(* IEC 61131-3 sources: volt/packages/volt-lsp-iec/test-corpus/pro2193/Device/Plc Logic/Application/09 Misc/Library Manager/L_MC1P_MotionControlBasic (part 6) *)

(* ---- L_MC1P_POSPROFILER.pou ---- *)
FUNCTION_BLOCK L_MC1P_POSPROFILER
VAR_INPUT
	XEXECUTE : BOOL := FALSE;
	XAUXEXECUTE : BOOL := FALSE;
	XABORT : BOOL := FALSE;
	XPOSMODE : BOOL := FALSE;
	ROVERRIDESPEED : LREAL := 1.0;
	ROVERRIDEACC : LREAL := 1.0;
	ROVERRIDEDEC : LREAL := 1.0;
	ROVERRIDEJERKACC : LREAL := 1.0;
	ROVERRIDEJERKDEC : LREAL := 1.0;
	LRACTPOS : LREAL := 0.0;
	LRACTSPEED : LREAL := 0.0;
	LRACTACC : LREAL := 0.0;
	LRTASKCYCLE : LREAL := 0.001;
	LRINVTASKCYCLE : LREAL := 1000.0;
	XCONTINUOUSUPDATE : BOOL;
	XWAIT : BOOL;
	LRCORRECTTIMEBASE : LREAL;
	WCALCPROFILEMODE : WORD;
	WSTRETCHPROFILEMODE : WORD := 0;
	XUSESTARTJERK : BOOL;
	LRSTARTJERK : LREAL;
	XUSEEXTERNPROFILECALCULATION : BOOL;
	ITFPOSPROFILECALCULATION : L_MC1P_IPosProfileCalculation;
	XINCREASEJERKDEC : BOOL;
	LRMAXJERKAPPL : LREAL;
END_VAR
VAR_OUTPUT
	XBUSY : BOOL;
	XDONE : BOOL;
	XABORTED : BOOL;
	XERROR : BOOL;
	LRSETPOS : LREAL;
	LRSETSPEED : LREAL;
	LRSETACC : LREAL;
	LRACTPROFILEJERK : LREAL;
	DWSTATE : DWORD;
	DWPROFILETYPE : DWORD;
	XNOPROFIEUPDATE : BOOL;
END_VAR
VAR_IN_OUT
	SCPROFILEPARAMETER : L_MC1P_ProfileParameter;
END_VAR
VAR
	SCPROFILEDATA : L_MC1P_ProfileData;
	XCALCPROFILEACTIVE : BOOL;
	LREVALTIME : LREAL;
	DWSTATEOFINTERPOLATOR : DWORD;
	XFLAGEXECUTE : BOOL;
	XFLAGAUXEXECUTE : BOOL;
	XFLAGABORT : BOOL;
	SCPROFILEPARAMETERINT : L_MC1P_ProfileParameter;
	SCPROFILEPARAMETEROLD : L_MC1P_ProfileParameter;
	ROVERRIDESPEEDOLD : LREAL;
	ROVERRIDEACCOLD : LREAL;
	ROVERRIDEDECOLD : LREAL;
	ROVERRIDEJERKACCOLD : LREAL;
	ROVERRIDEJERKDECOLD : LREAL;
	XSTARTCALCPROF : BOOL;
	XVELOVEREQZERO : BOOL;
	ARG1 : LREAL;
	XEXECUTEEDGE : BOOL;
	XAUXEXECUTEEDGE : BOOL;
	XABORTEDGE : BOOL;
	XCONTINUOUSUPDATEINT : BOOL;
	SCBUFFPROFILEPARAMETER : L_MC1P_ProfileParameter;
	SCBUFFPROFILEDATA : L_MC1P_ProfileData;
	XCALCULATEBUFFER : BOOL;
	XACITVATEBUFFERRANGE : BOOL;
	SCBUFFERDATAINT : L_MC1P_BufferData;
	LRTIMEACCBUFF : LREAL;
	XCALCPROFILEFIRSTCYCLEACTIVE : BOOL;
	WCALCPROFILESTEP : WORD;
	WITERATIONCYCLESLIMIT1 : WORD := 32;
	N : WORD;
	XSEARCHTIMESACTIVE : BOOL;
	XSEARCHTIMES1_DONE : BOOL;
	XCALCPROFILEDATAACTIVE : BOOL;
	XPROFILECALCULATED : BOOL;
	SIGNOFMAXVEL : LREAL;
	S_MIN : LREAL;
	DWMINPROFILETYPE : DWORD;
	VMAXMINTRIACC1 : LREAL;
	VMAXMINTRIACC2 : LREAL;
	LRRECIPRJERKACC : LREAL;
	LRRECIPRJERKDEC : LREAL;
	INITPROFILEDATA : L_MC1P_ProfileData;
	INITPHASEDATA : L_MC1P_ProfilePhaseData;
	INITINTPROFILEDATA : L_MC1P_IntProfileData;
	SCMINPOSPROFILEDATA : L_MC1P_IntProfileData;
	SCMINPROFILEDATA0 : L_MC1P_IntProfileData;
	SCMAXPROFILEDATA0 : L_MC1P_IntProfileData;
	SCMINPROFILEDATAINT : L_MC1P_IntProfileData;
	SCMINPROFILEDATA_ACC1 : L_MC1P_IntProfileDataAcc;
	SCMINPROFILEDATA_ACC2 : L_MC1P_IntProfileDataAcc;
	MINPROFILEDATA_PH57 : L_MC1P_IntProfileDataAcc;
	PROFILEPHASE : L_MC1P_ProfilePhaseData;
	JERKACCTEMP1 : LREAL;
	JERKACCTEMP2 : LREAL;
	VELPHASE4 : LREAL;
	MINVELPHASE4 : LREAL;
	PROVISIONALPROFILE : L_MC1P_IntProfileData;
	PROVISIONALPROFILEOLD : L_MC1P_IntProfileData;
	S_PROVISIONALPROFILE : LREAL;
	LRACTPROFILETIME : LREAL;
	T5_STARTVALUE : LREAL;
	T7_STARTVALUE : LREAL;
	T5_MAXVALUE : LREAL;
	T7_MAXVALUE : LREAL;
	T5_MINVALUE : LREAL;
	T7_MINVALUE : LREAL;
	MINPOSUNIT : LREAL;
	MINPOSUNITQUADRAT : LREAL;
	ESQR : LREAL;
	DT_AE : LREAL;
	DS_AE : LREAL;
	DT_A0 : LREAL;
	DS_A0 : LREAL;
	TMP : ARRAY [1..272] OF LREAL;
	INVJ : ARRAY [1..2, 1..2] OF LREAL;
	E : ARRAY [0..2] OF LREAL;
	P : ARRAY [1..2] OF LREAL;
	T5 : ARRAY [1..2] OF LREAL;
	LRMINREFJERK : LREAL;
	XPHASE0FINISHED : BOOL;
	LRSTARTACCINT : LREAL;
	LRSTARTVELINT : LREAL;
	LRSTARTPOSINT : LREAL;
	MAXPROFILEPHASEINDEX : WORD := 7;
	ALRPROFILEACC : ARRAY [0..8] OF LREAL;
	ALRPROFILEJERK : ARRAY [0..8] OF LREAL;
	ALRPROFILEPOS : ARRAY [0..8] OF LREAL;
	ALRPROFILETIME : ARRAY [0..8] OF LREAL;
	ALRPROFILEVEL : ARRAY [0..8] OF LREAL;
	REMAININGTIMEOFPROFILE : LREAL;
	REMAININGTIMEOFPROFILEAVAILABLE : BOOL;
END_VAR
END_FUNCTION_BLOCK

METHOD CALCPROFILEDATA
VAR_INPUT
	LRSTARTACC : LREAL;
	LRSTARTVEL : LREAL;
	LRSTARTPOS : LREAL;
	XVELMODE : BOOL;
END_VAR
VAR_OUTPUT
	XERROR : BOOL;
	DWSTATE : DWORD;
	DWPROFILETYPE : DWORD;
END_VAR
VAR_IN_OUT
	SCPROFILEDATA : L_MC1P_ProfileData;
	SCPROFILEPARAMETER : L_MC1P_ProfileParameter;
END_VAR
END_METHOD

METHOD CALCPROFILEDATACOMPLETE
VAR_INPUT
	LRSTARTACC : LREAL;
	LRSTARTVEL : LREAL;
	LRSTARTPOS : LREAL;
	XVELMODE : BOOL;
END_VAR
VAR_OUTPUT
	XERROR : BOOL;
	DWSTATE : DWORD;
	DWPROFILETYPE : DWORD;
END_VAR
VAR_IN_OUT
	SCPROFILEDATA : L_MC1P_ProfileData;
	SCPROFILEPARAMETER : L_MC1P_ProfileParameter;
END_VAR
END_METHOD

METHOD CALCSQRT : LREAL
VAR_INPUT
	ARG1 : LREAL;
END_VAR
END_METHOD

METHOD GETPROFILEIDXATPOS : WORD
VAR_INPUT
	LRPOS : LREAL;
END_VAR
VAR_IN_OUT
	SCPROFILEDATA : L_MC1P_ProfileData;
END_VAR
END_METHOD

METHOD GETSETVALUESNEXTCYCLE : BOOL
VAR_OUTPUT
	LRSETPOS : LREAL;
	LRSETSPEED : LREAL;
	LRSETACC : LREAL;
	DWSTATEOFINTERPOLATOR : DWORD;
END_VAR
END_METHOD

METHOD GETTIMEATPOS : LREAL
VAR_INPUT
	LRPOS : LREAL;
END_VAR
VAR_IN_OUT
	SCPROFILEDATA : L_MC1P_ProfileData;
END_VAR
END_METHOD

METHOD PROFILEINTERPOLATOR : BOOL
VAR_INPUT
	LREVALTIME : LREAL;
END_VAR
VAR_OUTPUT
	DWSTATE : DWORD;
	LRSETPOS : LREAL;
	LRSETVEL : LREAL;
	LRSETACC : LREAL;
END_VAR
VAR_IN_OUT
	SCPROFILEDATA : L_MC1P_ProfileData;
END_VAR
END_METHOD

METHOD REMAININGPROFILETIMEATPOS : BOOL
VAR_INPUT
	LRPROFILEPOS : LREAL;
END_VAR
VAR_OUTPUT
	LRREMAININGTIME : LREAL;
END_VAR
VAR_IN_OUT
	SCPROFILEDATA : L_MC1P_ProfileData;
END_VAR
END_METHOD

METHOD RESET
END_METHOD

METHOD RESETOUTPUT
END_METHOD

METHOD STRETCHPROFILE
VAR_INPUT
	LRTIMEBASE : LREAL;
END_VAR
VAR_IN_OUT
	SCPROFILEDATA : L_MC1P_ProfileData;
END_VAR
END_METHOD

METHOD FB_INIT : BOOL
VAR_INPUT
	BINITRETAINS : BOOL;
	BINCOPYCODE : BOOL;
END_VAR
END_METHOD

METHOD CALCULATEACCDIST : LREAL
VAR_INPUT
	LRACC : LREAL;
	LRJERK : LREAL;
	LRVEL : LREAL;
END_VAR
VAR_OUTPUT
	LRTIMEACC : LREAL;
END_VAR
END_METHOD

METHOD CALCULATEBUFFER : BOOL
VAR_INPUT
	LRACTPOS : LREAL;
	SCBUFFERDATA : L_MC1P_BufferData;
END_VAR
VAR_IN_OUT
	SCPROFILEPARAMETER : L_MC1P_ProfileParameter;
	SCPROFILEDATA : L_MC1P_ProfileData;
	SCBUFFPROFILEPARAMETER : L_MC1P_ProfileParameter;
	SCBUFFPROFILEDATA : L_MC1P_ProfileData;
END_VAR
END_METHOD

METHOD GETVELATPOS : LREAL
VAR_INPUT
	LRPOS : LREAL;
END_VAR
VAR_IN_OUT
	SCPROFILEDATA : L_MC1P_ProfileData;
END_VAR
END_METHOD

METHOD PROFILEINTERPOLATORBUFFER : BOOL
VAR_INPUT
	LREVALTIME : LREAL;
END_VAR
VAR_OUTPUT
	DWSTATE : DWORD;
	LRSETPOS : LREAL;
	LRSETVEL : LREAL;
	LRSETACC : LREAL;
END_VAR
VAR_IN_OUT
	SCPROFILEDATA1 : L_MC1P_ProfileData;
	SCPROFILEDATA2 : L_MC1P_ProfileData;
END_VAR
END_METHOD

METHOD SETBUFFERDATA
VAR_INPUT
	XENABLEBUFFER : BOOL;
	SCBUFFERDATA : L_MC1P_BufferData;
END_VAR
END_METHOD

METHOD CALCMINPOSUNIT : BOOL
VAR_INPUT
	SCMINPROFILEDATA : L_MC1P_IntProfileData;
	LRMAXVEL : LREAL;
	LRJERKACC1 : LREAL;
	LRMAXACC1 : LREAL;
	LRJERKACC2 : LREAL;
	LRMAXACC2 : LREAL;
	LRTARGETVEL : LREAL;
	LRTARGETACC : LREAL;
END_VAR
VAR_OUTPUT
	LRMINPOSUNIT : LREAL;
	LRMINVELUNIT : LREAL;
END_VAR
END_METHOD

METHOD CALCPROFILE : BOOL
VAR_INPUT
	DWPROFILETYPE : DWORD;
	LRSTARTACC : LREAL;
	LRSTARTVEL : LREAL;
	SCMINPROFILEDATA : L_MC1P_IntProfileData;
	SCMAXPROFILEDATA : L_MC1P_IntProfileData;
END_VAR
VAR_IN_OUT
	SCPROFILEPARAMETER : L_MC1P_ProfileParameter;
	SCPROFILEDATA : L_MC1P_ProfileData;
	WCHECKPROFILEMODE : WORD;
	DWSTATE : DWORD;
END_VAR
END_METHOD

METHOD CHECKPROFILEDATA
VAR_INPUT
	DWMODE : DWORD;
	LRTARGETPOS : LREAL;
	LRTARGETVEL : LREAL;
	LRTARGETACC : LREAL;
	LRJERKPHASE7 : LREAL;
END_VAR
VAR_OUTPUT
	XERROR : BOOL;
END_VAR
VAR_IN_OUT
	SCPROFILEDATA : L_MC1P_ProfileData;
END_VAR
END_METHOD

METHOD DEFPROFILEACCDEC
VAR_IN_OUT
	SCPROFILEPARAMETER : L_MC1P_ProfileParameter;
	LRSTARTACC : LREAL;
	LRSTARTVEL : LREAL;
	XVELMODE : BOOL;
END_VAR
END_METHOD

METHOD DEFPROFILEPHASE0 : BOOL
VAR_INPUT
	LRMINJERK : LREAL;
	XVELMODE : BOOL;
END_VAR
VAR_IN_OUT
	SCPROFILEPARAMETER : L_MC1P_ProfileParameter;
	LRSTARTACC : LREAL;
	LRSTARTVEL : LREAL;
	LRRECIPRJERKACC : LREAL;
	LRRECIPRJERKDEC : LREAL;
	SCPROFILEDATAPHASE0 : L_MC1P_ProfilePhaseData;
	SCMAXPROFILEDATA : L_MC1P_IntProfileData;
	SCMINPROFILEDATA : L_MC1P_IntProfileData;
	DWPROFILETYPE : DWORD;
	DWSTATE : DWORD;
END_VAR
END_METHOD

METHOD CALCMINPOSPROFILE : BOOL
VAR_INPUT
	MAXVEL : LREAL;
	MAXACC1 : LREAL;
	MAXACC2 : LREAL;
	JERKACC1 : LREAL;
	JERKACC2 : LREAL;
	MINJERK : LREAL;
	RECIPRJERKACC1 : LREAL;
	RECIPRJERKACC2 : LREAL;
	RECIPRMINJERK : LREAL;
	V0_ACC1 : LREAL;
	V0_ACC2 : LREAL;
	A0_ACC1 : LREAL;
	A0_ACC2 : LREAL;
	XVELMODE : BOOL;
END_VAR
VAR_IN_OUT
	DWMINPOSPROFILETYPE : DWORD;
	MINPOSPROFILEDATA : L_MC1P_IntProfileData;
	VMAXMINTRIACC1 : LREAL;
	VMAXMINTRIACC2 : LREAL;
END_VAR
END_METHOD

METHOD CALCMINPROFILE : BOOL
VAR_INPUT
	MAXVEL : LREAL;
	MAXACC1 : LREAL;
	MAXACC2 : LREAL;
	JERKACC1 : LREAL;
	JERKACC2 : LREAL;
	RECIPRJERKACC1 : LREAL;
	RECIPRJERKACC2 : LREAL;
	V0_ACC1 : LREAL;
	V0_ACC2 : LREAL;
	A0_ACC1 : LREAL;
	A0_ACC2 : LREAL;
	TARGETPOS : LREAL;
END_VAR
VAR_IN_OUT
	DWPROFILETYPE : DWORD;
	SCMINPROFILEDATA : L_MC1P_IntProfileData;
	SCMAXPROFILEDATA : L_MC1P_IntProfileData;
END_VAR
END_METHOD

METHOD CALCMINPROFILENEGACC : BOOL
VAR_INPUT
	V0 : LREAL;
	VE : LREAL;
	AMAX : LREAL;
	JERK : LREAL;
	JERKRECIPR : LREAL;
	A0 : LREAL;
	AE : LREAL;
END_VAR
VAR_OUTPUT
	DWPROFILETYPE : DWORD;
	PROFILEDATA_NEGACC : L_MC1P_IntProfileDataAcc;
END_VAR
END_METHOD

METHOD CALCMINPROFILENEGACCRND : BOOL
VAR_INPUT
	V0 : LREAL;
	VE : LREAL;
	AMAX : LREAL;
	JERK : LREAL;
	JERKRECIPR : LREAL;
	A0 : LREAL;
	AE : LREAL;
END_VAR
VAR_OUTPUT
	DWPROFILETYPE : DWORD;
	PROFILEDATA_NEGACC : L_MC1P_IntProfileDataAcc;
END_VAR
END_METHOD

METHOD CALCMINPROFILEPOSACC : BOOL
VAR_INPUT
	V0 : LREAL;
	VE : LREAL;
	AMAX : LREAL;
	A0 : LREAL;
	AE : LREAL;
	JERK : LREAL;
	JERKRECIPR : LREAL;
END_VAR
VAR_OUTPUT
	DWPROFILETYPE : DWORD;
	PROFILEDATA_POSACC : L_MC1P_IntProfileDataAcc;
END_VAR
END_METHOD

METHOD CALCMINTRI : BOOL
VAR_INPUT
	JERK : LREAL;
	RECIPRJERK : LREAL;
	A0 : LREAL;
	V0 : LREAL;
	MINCYCLETIME : LREAL;
END_VAR
VAR_OUTPUT
	VMAXMINTRIACC : LREAL;
	PROFILEDATA : L_MC1P_IntProfileDataAcc;
END_VAR
END_METHOD

METHOD CALCNEGPROFILEPHASE : BOOL
VAR_INPUT
	LRSTARTACC : LREAL;
	LRENDACC : LREAL;
	LRSTARTVEL : LREAL;
	LRJERK : LREAL;
	LRJERKRECIPR : LREAL;
	LRMINCYCLETIME : LREAL;
END_VAR
VAR_OUTPUT
	PROFILEPHASE : L_MC1P_ProfilePhaseData;
END_VAR
END_METHOD

METHOD CALCPROFILEPHASE : BOOL
VAR_INPUT
	LRSTARTACC : LREAL;
	LRENDACC : LREAL;
	LRSTARTVEL : LREAL;
	LRJERK : LREAL;
	LRJERKRECIPR : LREAL;
	LRMINCYCLETIME : LREAL;
END_VAR
VAR_OUTPUT
	PROFILEPHASE : L_MC1P_ProfilePhaseData;
END_VAR
END_METHOD

METHOD CALCPROVISIONALPROFILE
VAR_IN_OUT
	SCPROFILEPARAMETERINT : L_MC1P_ProfileParameter;
	LRSTARTVELINT : LREAL;
	LRSTARTACCINT : LREAL;
	LRRECIPRJERKACC : LREAL;
	LRRECIPRJERKDEC : LREAL;
	LRACTPROFILETIME : LREAL;
	XVELMODE : BOOL;
	SCPROVISIONALPROFILE : L_MC1P_IntProfileData;
END_VAR
END_METHOD

METHOD CALCPROVISIONALPROFILEDATA : BOOL
VAR_IN_OUT
	LRSTARTPOS : LREAL;
	LRSTARTVEL : LREAL;
	LRSTARTACC : LREAL;
	LRSTARTVELINT : LREAL;
	LRSTARTACCINT : LREAL;
	LRRECIPRJERKACC : LREAL;
	LRRECIPRJERKDEC : LREAL;
	SCPROFILEPARAMETERINT : L_MC1P_ProfileParameter;
	XVELMODE : BOOL;
	SIGNOFMAXVEL : LREAL;
	DWPROFILETYPE : DWORD;
	DWMINPOSPROFILETYPE : DWORD;
	XCALCPROFILE : BOOL;
	WCALCPROFILESTEP : WORD;
	XPOSITIVEMOVEMENT : BOOL;
	SCPROFILEDATAPHASE0 : L_MC1P_ProfilePhaseData;
	SCPROFILEDATA : L_MC1P_ProfileData;
	DWSTATECALCPROFILE : DWORD;
	SCMAXPROFILEDATA : L_MC1P_IntProfileData;
	SCMINPROFILEDATA : L_MC1P_IntProfileData;
END_VAR
END_METHOD

METHOD CALCREVPROFILE : BOOL
VAR_INPUT
	V0 : LREAL;
	VE : LREAL;
	AMAX : LREAL;
	A0 : LREAL;
	AE : LREAL;
	JERK : LREAL;
	JERKRECIPR : LREAL;
END_VAR
VAR_OUTPUT
	DWPROFILETYPE : DWORD;
	PROFILEDATA_POSACC : L_MC1P_IntProfileDataAcc;
END_VAR
END_METHOD

METHOD CALCVELPROFILEPHASE : BOOL
VAR_INPUT
	LRSTARTACC : LREAL;
	LRENDACC : LREAL;
	LRSTARTVEL : LREAL;
	LRJERK : LREAL;
	LRJERKRECIPR : LREAL;
	LRMINCYCLETIME : LREAL;
END_VAR
VAR_OUTPUT
	PROFILEPHASE : L_MC1P_ProfilePhaseData;
END_VAR
END_METHOD

METHOD IDENTINCRJERKPROFILE : BOOL
VAR_INPUT
	MINPROFILETYPE : DWORD;
	MAXACC2 : LREAL;
	MAXJERK : LREAL;
	V0_ACC1 : LREAL;
	V0_ACC2 : LREAL;
	A0_ACC1 : LREAL;
	A0_ACC2 : LREAL;
	TARGETPOS : LREAL;
END_VAR
VAR_OUTPUT
	DWINCRJERKPROFILETYPE : DWORD;
END_VAR
VAR_IN_OUT
	JERKACC2 : LREAL;
	RECIPRJERKACC2 : LREAL;
	SCMAXPROFILEDATA : L_MC1P_IntProfileData;
	SCMINPROFILEDATA : L_MC1P_IntProfileData;
END_VAR
END_METHOD

METHOD IDENTMINNEGPROFILE : BOOL
VAR_INPUT
	MINPROFILETYPE : DWORD;
	MAXVEL : LREAL;
	MAXACC : LREAL;
	JERK : LREAL;
	RECIPRJERK : LREAL;
	V0_ACC1 : LREAL;
	V0_ACC2 : LREAL;
	A0_ACC1 : LREAL;
	A0_ACC2 : LREAL;
	TARGETPOS : LREAL;
END_VAR
VAR_OUTPUT
	DWPROFILETYPE : DWORD;
END_VAR
VAR_IN_OUT
	SCMAXPROFILEDATA : L_MC1P_IntProfileData;
	SCMINPROFILEDATA : L_MC1P_IntProfileData;
END_VAR
END_METHOD

METHOD IDENTMINNEGPROFILE_A0EQ0_AENE0
VAR_INPUT
	MAXVEL : LREAL;
	SIGNOFMAXVEL : LREAL;
	MAXACC : LREAL;
	JERK : LREAL;
	RECIPRJERK : LREAL;
	V0_ACC1 : LREAL;
	V0_ACC2 : LREAL;
	A0_ACC1 : LREAL;
	A0_ACC2 : LREAL;
	TARGETPOS : LREAL;
	TARGETPOSTOLERANCE : LREAL;
END_VAR
VAR_OUTPUT
	DWPROFILETYPE : DWORD;
END_VAR
VAR_IN_OUT
	SCMAXPROFILEDATA : L_MC1P_IntProfileData;
	SCMINPROFILEDATA : L_MC1P_IntProfileData;
END_VAR
END_METHOD

METHOD IDENTMINNEGPROFILE_AENE0
VAR_INPUT
	MAXVEL : LREAL;
	SIGNOFMAXVEL : LREAL;
	MAXACC : LREAL;
	JERK : LREAL;
	RECIPRJERK : LREAL;
	V0_ACC1 : LREAL;
	V0_ACC2 : LREAL;
	A0_ACC1 : LREAL;
	A0_ACC2 : LREAL;
	TARGETPOS : LREAL;
	TARGETPOSTOLERANCE : LREAL;
END_VAR
VAR_IN_OUT
	SCMAXPROFILEDATA : L_MC1P_IntProfileData;
	SCMINPROFILEDATA : L_MC1P_IntProfileData;
	DWPROFILETYPE : DWORD;
END_VAR
END_METHOD

METHOD IDENTMINPOSPROFILE_AENE0
VAR_INPUT
	MAXVEL : LREAL;
	SIGNOFMAXVEL : LREAL;
	MAXACC : LREAL;
	JERK : LREAL;
	RECIPRJERK : LREAL;
	V0_ACC1 : LREAL;
	V0_ACC2 : LREAL;
	A0_ACC1 : LREAL;
	A0_ACC2 : LREAL;
	TARGETPOS : LREAL;
	TARGETPOSTOLERANCE : LREAL;
END_VAR
VAR_IN_OUT
	SCMAXPROFILEDATA : L_MC1P_IntProfileData;
	SCMINPROFILEDATA : L_MC1P_IntProfileData;
	DWPROFILETYPE : DWORD;
END_VAR
END_METHOD

METHOD IDENTMINPROFILE : BOOL
VAR_INPUT
	MAXVEL : LREAL;
	MAXACC1 : LREAL;
	MAXACC2 : LREAL;
	MINJERK : LREAL;
	RECIPRMINJERK : LREAL;
	V0_ACC1 : LREAL;
	A0_ACC1 : LREAL;
	TARGETPOS : LREAL;
	XVELMODE : BOOL;
END_VAR
VAR_IN_OUT
	DWPROFILETYPE : DWORD;
	SCMAXPROFILEDATA : L_MC1P_IntProfileData;
	SCMINPROFILEDATA : L_MC1P_IntProfileData;
	DWMINPROFILETYPE : DWORD;
	V0_ACC2 : LREAL;
	A0_ACC2 : LREAL;
	JERKACC1 : LREAL;
	JERKACC2 : LREAL;
	RECIPRJERKACC1 : LREAL;
	RECIPRJERKACC2 : LREAL;
	DWSTATE : DWORD;
END_VAR
END_METHOD

METHOD IDENTPROFILETYPE : DWORD
VAR_INPUT
	XVELMODE : BOOL;
	LRSTARTVEL : LREAL;
	LRSTARTACC : LREAL;
END_VAR
VAR_IN_OUT
	SCPROFILEPARAMETER : L_MC1P_ProfileParameter;
	DWPROFILETYPE : DWORD;
	SCMINPROFILEDATA : L_MC1P_IntProfileData;
	SCMAXPROFILEDATA : L_MC1P_IntProfileData;
	DWSTATE : DWORD;
END_VAR
END_METHOD

METHOD IDENTSIMPLEPROFILE
VAR_INPUT
	DWMINPOSPROFILETYPE : DWORD;
	VMAXMINTRIACC1 : LREAL;
	VMAXMINTRIACC2 : LREAL;
	MAXACC1 : LREAL;
	MAXACC2 : LREAL;
	JERKACC1 : LREAL;
	JERKACC2 : LREAL;
	V0_ACC1 : LREAL;
	A0_ACC1 : LREAL;
	RECIPRJERKACC1 : LREAL;
	RECIPRJERKACC2 : LREAL;
	LRTARGETPOS : LREAL;
	SIGNOFMAXVEL : LREAL;
END_VAR
VAR_OUTPUT
	DWPROFILETYPE : DWORD;
END_VAR
VAR_IN_OUT
	SCMINPROFILEDATA : L_MC1P_IntProfileData;
	SCMAXPROFILEDATA : L_MC1P_IntProfileData;
	V0_ACC2 : LREAL;
	A0_ACC2 : LREAL;
END_VAR
END_METHOD

METHOD IDENTSIMPLETRAPNEG : BOOL
VAR_INPUT
	MAXACC2 : LREAL;
	V0_ACC1 : LREAL;
	V0_ACC2 : LREAL;
	A0_ACC1 : LREAL;
	A0_ACC2 : LREAL;
	JERKACC1 : LREAL;
	JERKACC2 : LREAL;
	RECIPRJERKACC2 : LREAL;
	TARGETPOS : LREAL;
	SIGNOFMAXVEL : LREAL;
END_VAR
VAR_OUTPUT
	DWPROFILETYPE : DWORD;
END_VAR
VAR_IN_OUT
	SCMINPROFILEDATA : L_MC1P_IntProfileData;
	SCMAXPROFILEDATA : L_MC1P_IntProfileData;
END_VAR
END_METHOD

METHOD IDENTSIMPLETRAPPOS : BOOL
VAR_INPUT
	MAXACC1 : LREAL;
	V0_ACC1 : LREAL;
	V0_ACC2 : LREAL;
	A0_ACC1 : LREAL;
	A0_ACC2 : LREAL;
	JERKACC1 : LREAL;
	JERKACC2 : LREAL;
	RECIPRJERKACC1 : LREAL;
	TARGETPOS : LREAL;
	SIGNOFMAXVEL : LREAL;
END_VAR
VAR_OUTPUT
	DWPROFILETYPE : DWORD;
END_VAR
VAR_IN_OUT
	SCMINPROFILEDATA : L_MC1P_IntProfileData;
	SCMAXPROFILEDATA : L_MC1P_IntProfileData;
END_VAR
END_METHOD

METHOD IDENTSIMPLETRAPPOSTRINEG : BOOL
VAR_INPUT
	MAXACC1 : LREAL;
	JERKACC1 : LREAL;
	RECIPRJERKACC1 : LREAL;
	V0_ACC1 : LREAL;
	A0_ACC1 : LREAL;
	VMAXACC1 : LREAL;
	VMAXACC2 : LREAL;
	JERKACC2 : LREAL;
	TARGETPOS : LREAL;
	SIGNOFMAXVEL : LREAL;
END_VAR
VAR_OUTPUT
	DWPROFILETYPE : DWORD;
END_VAR
VAR_IN_OUT
	SCMINPROFILEDATA : L_MC1P_IntProfileData;
	SCMAXPROFILEDATA : L_MC1P_IntProfileData;
END_VAR
END_METHOD

METHOD IDENTSIMPLETRINEG : BOOL
VAR_INPUT
	V0_ACC1 : LREAL;
	A0_ACC1 : LREAL;
	A0_ACC2 : LREAL;
	JERKACC1 : LREAL;
	JERKACC2 : LREAL;
	RECIPRJERKACC2 : LREAL;
	TARGETPOS : LREAL;
	SIGNOFMAXVEL : LREAL;
END_VAR
VAR_OUTPUT
	DWPROFILETYPE : DWORD;
END_VAR
VAR_IN_OUT
	SCMINPROFILEDATA : L_MC1P_IntProfileData;
	SCMAXPROFILEDATA : L_MC1P_IntProfileData;
END_VAR
END_METHOD

METHOD IDENTSIMPLETRIPOS : BOOL
VAR_INPUT
	V0_ACC1 : LREAL;
	A0_ACC1 : LREAL;
	A0_ACC2 : LREAL;
	JERKACC1 : LREAL;
	JERKACC2 : LREAL;
	RECIPRJERKACC1 : LREAL;
	TARGETPOS : LREAL;
	SIGNOFMAXVEL : LREAL;
END_VAR
VAR_OUTPUT
	DWPROFILETYPE : DWORD;
END_VAR
VAR_IN_OUT
	SCMINPROFILEDATA : L_MC1P_IntProfileData;
	SCMAXPROFILEDATA : L_MC1P_IntProfileData;
END_VAR
END_METHOD

METHOD IDENTSIMPLETRIPOSTRAPNEG : BOOL
VAR_INPUT
	V0_ACC1 : LREAL;
	A0_ACC1 : LREAL;
	MAXACC2 : LREAL;
	JERKACC2 : LREAL;
	RECIPRJERKACC2 : LREAL;
	V0_ACC2 : LREAL;
	A0_ACC2 : LREAL;
	VMAXMINTRIACC1 : LREAL;
	JERKACC1 : LREAL;
	RECIPRJERKACC1 : LREAL;
	TARGETPOS : LREAL;
	SIGNOFMAXVEL : LREAL;
END_VAR
VAR_OUTPUT
	DWPROFILETYPE : DWORD;
END_VAR
VAR_IN_OUT
	SCMINPROFILEDATA : L_MC1P_IntProfileData;
	SCMAXPROFILEDATA : L_MC1P_IntProfileData;
END_VAR
END_METHOD

METHOD IDENTSIMPLETRIPOSTRINEG : BOOL
VAR_INPUT
	V0_ACC1 : LREAL;
	A0_ACC1 : LREAL;
	AMAX : LREAL;
	RECIPRJERKACC1 : LREAL;
	JERKACC1 : LREAL;
	JERKACC2 : LREAL;
	TARGETPOS : LREAL;
	VMAXACC1 : LREAL;
	VMAXACC2 : LREAL;
	SIGNOFMAXVEL : LREAL;
END_VAR
VAR_OUTPUT
	DWPROFILETYPE : DWORD;
END_VAR
VAR_IN_OUT
	SCMINPROFILEDATA : L_MC1P_IntProfileData;
	SCMAXPROFILEDATA : L_MC1P_IntProfileData;
END_VAR
END_METHOD

METHOD CALCPROFILE_10X0_30X0 : BOOL
VAR_INPUT
	LRSTARTACC : LREAL;
	LRSTARTVEL : LREAL;
	LRMAXACC : LREAL;
	LRMAXDEC : LREAL;
	LRMAXVEL : LREAL;
	LRTARGETACC : LREAL;
	LRTARGETVEL : LREAL;
	LRTARGETPOS : LREAL;
	LRJERKACC : LREAL;
	LRJERKDEC : LREAL;
	LRJERKTIMEACC : LREAL;
	LRJERKTIMEDEC : LREAL;
	SCMINPROFILEDATA : L_MC1P_IntProfileData;
	SCMAXPROFILEDATA : L_MC1P_IntProfileData;
END_VAR
VAR_OUTPUT
	DWSTATE : DWORD;
END_VAR
VAR_IN_OUT
	SCPROFILEDATA : L_MC1P_ProfileData;
	SCPROFILEPARAMETER : L_MC1P_ProfileParameter;
END_VAR
END_METHOD

METHOD CALCPROFILE_20CB : BOOL
VAR_INPUT
	LRSTARTACC : LREAL;
	LRSTARTVEL : LREAL;
	LRMAXACC : LREAL;
	LRMAXDEC : LREAL;
	LRMAXVEL : LREAL;
	LRTARGETACC : LREAL;
	LRTARGETVEL : LREAL;
	LRTARGETPOS : LREAL;
	LRJERKACC : LREAL;
	LRJERKDEC : LREAL;
	LRJERKTIMEACC : LREAL;
	LRJERKTIMEDEC : LREAL;
	SCMAXPROFILEDATA : L_MC1P_IntProfileData;
	SCMINPROFILEDATA : L_MC1P_IntProfileData;
END_VAR
VAR_OUTPUT
	DWSTATE : DWORD;
END_VAR
VAR_IN_OUT
	SCPROFILEDATA : L_MC1P_ProfileData;
	SCPROFILEPARAMETER : L_MC1P_ProfileParameter;
END_VAR
END_METHOD

METHOD CALCPROFILE_20CB_LINVELPH57_NEG : BOOL
VAR_INPUT
	LRSTARTACC : LREAL;
	LRSTARTVEL : LREAL;
	LRMAXACC : LREAL;
	LRMAXDEC : LREAL;
	LRMAXVEL : LREAL;
	LRTARGETACC : LREAL;
	LRTARGETVEL : LREAL;
	LRTARGETPOS : LREAL;
	LRJERKACC : LREAL;
	LRJERKDEC : LREAL;
	LRJERKTIMEACC : LREAL;
	LRJERKTIMEDEC : LREAL;
	T7 : LREAL;
END_VAR
VAR_IN_OUT
	SCPROFILEDATA : L_MC1P_ProfileData;
END_VAR
END_METHOD

METHOD CALCPROFILE_20CB_LINVELPH57_POS : BOOL
VAR_INPUT
	LRSTARTACC : LREAL;
	LRSTARTVEL : LREAL;
	LRMAXACC : LREAL;
	LRMAXDEC : LREAL;
	LRMAXVEL : LREAL;
	LRTARGETACC : LREAL;
	LRTARGETVEL : LREAL;
	LRTARGETPOS : LREAL;
	LRJERKACC : LREAL;
	LRJERKDEC : LREAL;
	LRJERKTIMEACC : LREAL;
	LRJERKTIMEDEC : LREAL;
	T7 : LREAL;
END_VAR
VAR_IN_OUT
	SCPROFILEDATA : L_MC1P_ProfileData;
END_VAR
END_METHOD

METHOD CALCPROFILE_20CB_AOGEAMAX_PROFILEDATA : BOOL
VAR_INPUT
	LRSTARTACC : LREAL;
	LRSTARTVEL : LREAL;
	LRMAXACC : LREAL;
	LRMAXDEC : LREAL;
	LRMAXVEL : LREAL;
	LRTARGETACC : LREAL;
	LRTARGETVEL : LREAL;
	LRTARGETPOS : LREAL;
	LRJERKACC : LREAL;
	LRJERKDEC : LREAL;
	LRJERKTIMEACC : LREAL;
	LRJERKTIMEDEC : LREAL;
	T7 : LREAL;
END_VAR
VAR_IN_OUT
	SCPROFILEDATA : L_MC1P_ProfileData;
END_VAR
END_METHOD

METHOD CALCPROFILE_20CB_AOGEAMAX_SEARCHTIMES : BOOL
VAR_INPUT
	LRSTARTACC : LREAL;
	LRSTARTVEL : LREAL;
	LRMAXACC : LREAL;
	LRMAXDEC : LREAL;
	LRMAXVEL : LREAL;
	LRTARGETACC : LREAL;
	LRTARGETVEL : LREAL;
	LRTARGETPOS : LREAL;
	LRJERKACC : LREAL;
	LRJERKDEC : LREAL;
	LRJERKTIMEACC : LREAL;
	LRJERKTIMEDEC : LREAL;
	T7_MINVALUE : LREAL;
	T7_MAXVALUE : LREAL;
END_VAR
VAR_IN_OUT
	T7 : LREAL;
END_VAR
END_METHOD

METHOD CALCPROFILE_20D1 : BOOL
VAR_INPUT
	LRSTARTACC : LREAL;
	LRSTARTVEL : LREAL;
	LRMAXACC : LREAL;
	LRMAXDEC : LREAL;
	LRMAXVEL : LREAL;
	LRTARGETACC : LREAL;
	LRTARGETVEL : LREAL;
	LRTARGETPOS : LREAL;
	LRJERKACC : LREAL;
	LRJERKDEC : LREAL;
	LRJERKTIMEACC : LREAL;
	LRJERKTIMEDEC : LREAL;
	SCMAXPROFILEDATA : L_MC1P_IntProfileData;
	SCMINPROFILEDATA : L_MC1P_IntProfileData;
END_VAR
VAR_OUTPUT
	DWSTATE : DWORD;
END_VAR
VAR_IN_OUT
	SCPROFILEDATA : L_MC1P_ProfileData;
END_VAR
END_METHOD

METHOD CALCPROFILE_20D1_PROFILEDATA : BOOL
VAR_INPUT
	LRSTARTACC : LREAL;
	LRSTARTVEL : LREAL;
	LRMAXACC : LREAL;
	LRMAXDEC : LREAL;
	LRMAXVEL : LREAL;
	LRTARGETACC : LREAL;
	LRTARGETVEL : LREAL;
	LRTARGETPOS : LREAL;
	LRJERKACC : LREAL;
	LRJERKDEC : LREAL;
	LRJERKTIMEACC : LREAL;
	LRJERKTIMEDEC : LREAL;
	T7 : LREAL;
END_VAR
VAR_IN_OUT
	SCPROFILEDATA : L_MC1P_ProfileData;
END_VAR
END_METHOD

METHOD CALCPROFILE_20D1_SEARCHTIMES : BOOL
VAR_INPUT
	LRSTARTACC : LREAL;
	LRSTARTVEL : LREAL;
	LRMAXACC : LREAL;
	LRMAXDEC : LREAL;
	LRMAXVEL : LREAL;
	LRTARGETACC : LREAL;
	LRTARGETVEL : LREAL;
	LRTARGETPOS : LREAL;
	LRJERKACC : LREAL;
	LRJERKDEC : LREAL;
	LRJERKTIMEACC : LREAL;
	LRJERKTIMEDEC : LREAL;
	T7_MINVALUE : LREAL;
	T7_MAXVALUE : LREAL;
END_VAR
VAR_IN_OUT
	T7 : LREAL;
END_VAR
END_METHOD

METHOD CALCPROFILE_20DB : BOOL
VAR_INPUT
	LRSTARTACC : LREAL;
	LRSTARTVEL : LREAL;
	LRMAXACC : LREAL;
	LRMAXDEC : LREAL;
	LRMAXVEL : LREAL;
	LRTARGETACC : LREAL;
	LRTARGETVEL : LREAL;
	LRTARGETPOS : LREAL;
	LRJERKACC : LREAL;
	LRJERKDEC : LREAL;
	LRJERKTIMEACC : LREAL;
	LRJERKTIMEDEC : LREAL;
	SCMAXPROFILEDATA : L_MC1P_IntProfileData;
	SCMINPROFILEDATA : L_MC1P_IntProfileData;
END_VAR
VAR_OUTPUT
	DWSTATE : DWORD;
END_VAR
VAR_IN_OUT
	SCPROFILEDATA : L_MC1P_ProfileData;
	SCPROFILEPARAMETER : L_MC1P_ProfileParameter;
END_VAR
END_METHOD

METHOD CALCPROFILE_20DB_PROFILEDATA : BOOL
VAR_INPUT
	LRSTARTACC : LREAL;
	LRSTARTVEL : LREAL;
	LRMAXACC : LREAL;
	LRMAXDEC : LREAL;
	LRMAXVEL : LREAL;
	LRTARGETACC : LREAL;
	LRTARGETVEL : LREAL;
	LRTARGETPOS : LREAL;
	LRJERKACC : LREAL;
	LRJERKDEC : LREAL;
	LRJERKTIMEACC : LREAL;
	LRJERKTIMEDEC : LREAL;
	T7 : LREAL;
END_VAR
VAR_IN_OUT
	SCPROFILEDATA : L_MC1P_ProfileData;
END_VAR
END_METHOD

METHOD CALCPROFILE_20DB_SEARCHTIMES : BOOL
VAR_INPUT
	LRSTARTACC : LREAL;
	LRSTARTVEL : LREAL;
	LRMAXACC : LREAL;
	LRMAXDEC : LREAL;
	LRMAXVEL : LREAL;
	LRTARGETACC : LREAL;
	LRTARGETVEL : LREAL;
	LRTARGETPOS : LREAL;
	LRJERKACC : LREAL;
	LRJERKDEC : LREAL;
	LRJERKTIMEACC : LREAL;
	LRJERKTIMEDEC : LREAL;
	T7_MINVALUE : LREAL;
	T7_MAXVALUE : LREAL;
END_VAR
VAR_IN_OUT
	T7 : LREAL;
END_VAR
END_METHOD

METHOD CALCPROFILE_40A0 : BOOL
VAR_INPUT
	LRSTARTACC : LREAL;
	LRSTARTVEL : LREAL;
	LRMAXACC : LREAL;
	LRMAXDEC : LREAL;
	LRMAXVEL : LREAL;
	LRTARGETACC : LREAL;
	LRTARGETVEL : LREAL;
	LRTARGETPOS : LREAL;
	LRJERKACC : LREAL;
	LRJERKDEC : LREAL;
	LRJERKTIMEACC : LREAL;
	LRJERKTIMEDEC : LREAL;
END_VAR
VAR_OUTPUT
	DWSTATE : DWORD;
END_VAR
VAR_IN_OUT
	SCPROFILEDATA : L_MC1P_ProfileData;
	SCPROFILEPARAMETER : L_MC1P_ProfileParameter;
END_VAR
END_METHOD

METHOD CALCPROFILE_40A0_LINVELPH1357_NEG : BOOL
VAR_INPUT
	LRSTARTACC : LREAL;
	LRSTARTVEL : LREAL;
	LRMAXACC : LREAL;
	LRMAXDEC : LREAL;
	LRMAXVEL : LREAL;
	LRTARGETACC : LREAL;
	LRTARGETVEL : LREAL;
	LRTARGETPOS : LREAL;
	LRJERKACC : LREAL;
	LRJERKDEC : LREAL;
	LRJERKTIMEACC : LREAL;
	LRJERKTIMEDEC : LREAL;
END_VAR
VAR_IN_OUT
	SCPROFILEDATA : L_MC1P_ProfileData;
END_VAR
END_METHOD

METHOD CALCPROFILE_40A0_LINVELPH1357_POS : BOOL
VAR_INPUT
	LRSTARTACC : LREAL;
	LRSTARTVEL : LREAL;
	LRMAXACC : LREAL;
	LRMAXDEC : LREAL;
	LRMAXVEL : LREAL;
	LRTARGETACC : LREAL;
	LRTARGETVEL : LREAL;
	LRTARGETPOS : LREAL;
	LRJERKACC : LREAL;
	LRJERKDEC : LREAL;
	LRJERKTIMEACC : LREAL;
	LRJERKTIMEDEC : LREAL;
END_VAR
VAR_IN_OUT
	SCPROFILEDATA : L_MC1P_ProfileData;
END_VAR
END_METHOD

METHOD CALCPROFILE_40A0_LINVELPH13_NEG : BOOL
VAR_INPUT
	LRSTARTACC : LREAL;
	LRSTARTVEL : LREAL;
	LRMAXACC : LREAL;
	LRMAXDEC : LREAL;
	LRMAXVEL : LREAL;
	LRTARGETACC : LREAL;
	LRTARGETVEL : LREAL;
	LRTARGETPOS : LREAL;
	LRJERKACC : LREAL;
	LRJERKDEC : LREAL;
	LRJERKTIMEACC : LREAL;
	LRJERKTIMEDEC : LREAL;
END_VAR
VAR_IN_OUT
	SCPROFILEDATA : L_MC1P_ProfileData;
END_VAR
END_METHOD

METHOD CALCPROFILE_40A0_LINVELPH13_POS : BOOL
VAR_INPUT
	LRSTARTACC : LREAL;
	LRSTARTVEL : LREAL;
	LRMAXACC : LREAL;
	LRMAXDEC : LREAL;
	LRMAXVEL : LREAL;
	LRTARGETACC : LREAL;
	LRTARGETVEL : LREAL;
	LRTARGETPOS : LREAL;
	LRJERKACC : LREAL;
	LRJERKDEC : LREAL;
	LRJERKTIMEACC : LREAL;
	LRJERKTIMEDEC : LREAL;
END_VAR
VAR_IN_OUT
	SCPROFILEDATA : L_MC1P_ProfileData;
END_VAR
END_METHOD

METHOD CALCPROFILE_40A0_LINVELPH57_NEG : BOOL
VAR_INPUT
	LRSTARTACC : LREAL;
	LRSTARTVEL : LREAL;
	LRMAXACC : LREAL;
	LRMAXDEC : LREAL;
	LRMAXVEL : LREAL;
	LRTARGETACC : LREAL;
	LRTARGETVEL : LREAL;
	LRTARGETPOS : LREAL;
	LRJERKACC : LREAL;
	LRJERKDEC : LREAL;
	LRJERKTIMEACC : LREAL;
	LRJERKTIMEDEC : LREAL;
END_VAR
VAR_IN_OUT
	SCPROFILEDATA : L_MC1P_ProfileData;
END_VAR
END_METHOD

METHOD CALCPROFILE_40A0_LINVELPH57_POS : BOOL
VAR_INPUT
	LRSTARTACC : LREAL;
	LRSTARTVEL : LREAL;
	LRMAXACC : LREAL;
	LRMAXDEC : LREAL;
	LRMAXVEL : LREAL;
	LRTARGETACC : LREAL;
	LRTARGETVEL : LREAL;
	LRTARGETPOS : LREAL;
	LRJERKACC : LREAL;
	LRJERKDEC : LREAL;
	LRJERKTIMEACC : LREAL;
	LRJERKTIMEDEC : LREAL;
END_VAR
VAR_IN_OUT
	SCPROFILEDATA : L_MC1P_ProfileData;
END_VAR
END_METHOD

METHOD CALCPROFILE_40A0_A0LTAMAX_NEG : BOOL
VAR_INPUT
	LRSTARTACC : LREAL;
	LRSTARTVEL : LREAL;
	LRMAXACC : LREAL;
	LRMAXDEC : LREAL;
	LRMAXVEL : LREAL;
	LRTARGETACC : LREAL;
	LRTARGETVEL : LREAL;
	LRTARGETPOS : LREAL;
	LRJERKACC : LREAL;
	LRJERKDEC : LREAL;
	LRJERKTIMEACC : LREAL;
	LRJERKTIMEDEC : LREAL;
END_VAR
VAR_IN_OUT
	SCPROFILEDATA : L_MC1P_ProfileData;
END_VAR
END_METHOD

METHOD CALCPROFILE_40A0_A0LTAMAX_POS : BOOL
VAR_INPUT
	LRSTARTACC : LREAL;
	LRSTARTVEL : LREAL;
	LRMAXACC : LREAL;
	LRMAXDEC : LREAL;
	LRMAXVEL : LREAL;
	LRTARGETACC : LREAL;
	LRTARGETVEL : LREAL;
	LRTARGETPOS : LREAL;
	LRJERKACC : LREAL;
	LRJERKDEC : LREAL;
	LRJERKTIMEACC : LREAL;
	LRJERKTIMEDEC : LREAL;
END_VAR
VAR_IN_OUT
	SCPROFILEDATA : L_MC1P_ProfileData;
END_VAR
END_METHOD

METHOD CALCPROFILE_40B0 : BOOL
VAR_INPUT
	LRSTARTACC : LREAL;
	LRSTARTVEL : LREAL;
	LRMAXACC : LREAL;
	LRMAXDEC : LREAL;
	LRMAXVEL : LREAL;
	LRTARGETACC : LREAL;
	LRTARGETVEL : LREAL;
	LRTARGETPOS : LREAL;
	LRJERKACC : LREAL;
	LRJERKDEC : LREAL;
	LRJERKTIMEACC : LREAL;
	LRJERKTIMEDEC : LREAL;
	SCMAXPROFILEDATA : L_MC1P_IntProfileData;
	SCMINPROFILEDATA : L_MC1P_IntProfileData;
END_VAR
VAR_OUTPUT
	DWSTATE : DWORD;
END_VAR
VAR_IN_OUT
	SCPROFILEDATA : L_MC1P_ProfileData;
	SCPROFILEPARAMETER : L_MC1P_ProfileParameter;
END_VAR
END_METHOD

METHOD CALCPROFILE_40B0_LINVELPH13 : BOOL
VAR_INPUT
	LRSTARTACC : LREAL;
	LRSTARTVEL : LREAL;
	LRMAXACC : LREAL;
	LRMAXDEC : LREAL;
	LRMAXVEL : LREAL;
	LRTARGETACC : LREAL;
	LRTARGETVEL : LREAL;
	LRTARGETPOS : LREAL;
	LRJERKACC : LREAL;
	LRJERKDEC : LREAL;
	LRJERKTIMEACC : LREAL;
	LRJERKTIMEDEC : LREAL;
	T5 : LREAL;
	T7 : LREAL;
END_VAR
VAR_IN_OUT
	SCPROFILEDATA : L_MC1P_ProfileData;
END_VAR
END_METHOD

METHOD CALCPROFILE_40B0_LINVELPH13_SEARCHTIMEST5T7 : BOOL
VAR_INPUT
	LRSTARTACC : LREAL;
	LRSTARTVEL : LREAL;
	LRMAXACC : LREAL;
	LRMAXDEC : LREAL;
	LRMAXVEL : LREAL;
	LRTARGETACC : LREAL;
	LRTARGETVEL : LREAL;
	LRTARGETPOS : LREAL;
	LRMINPOSUNIT : LREAL;
	LRJERKACC : LREAL;
	LRJERKDEC : LREAL;
	LRJERKTIMEACC : LREAL;
	LRJERKTIMEDEC : LREAL;
	T5_STARTVALUE : LREAL;
	T7_STARTVALUE : LREAL;
END_VAR
VAR_IN_OUT
	T5 : LREAL;
	T7 : LREAL;
END_VAR
END_METHOD

METHOD CALCPROFILE_40B0_A0LTAMAXSEARCHTIMEST5T7 : BOOL
VAR_INPUT
	LRSTARTACC : LREAL;
	LRSTARTVEL : LREAL;
	LRMAXACC : LREAL;
	LRMAXDEC : LREAL;
	LRMAXVEL : LREAL;
	LRTARGETACC : LREAL;
	LRTARGETVEL : LREAL;
	LRTARGETPOS : LREAL;
	LRMINPOSUNIT : LREAL;
	LRJERKACC : LREAL;
	LRJERKDEC : LREAL;
	LRJERKTIMEACC : LREAL;
	LRJERKTIMEDEC : LREAL;
	T5_STARTVALUE : LREAL;
	T7_STARTVALUE : LREAL;
END_VAR
VAR_IN_OUT
	T5 : LREAL;
	T7 : LREAL;
END_VAR
END_METHOD

METHOD CALCPROFILE_40B0_A0LTAMAXT5T7 : BOOL
VAR_INPUT
	LRSTARTACC : LREAL;
	LRSTARTVEL : LREAL;
	LRMAXACC : LREAL;
	LRMAXDEC : LREAL;
	LRMAXVEL : LREAL;
	LRTARGETACC : LREAL;
	LRTARGETVEL : LREAL;
	LRTARGETPOS : LREAL;
	LRJERKACC : LREAL;
	LRJERKDEC : LREAL;
	LRJERKTIMEACC : LREAL;
	LRJERKTIMEDEC : LREAL;
	T5 : LREAL;
	T7 : LREAL;
END_VAR
VAR_IN_OUT
	SCPROFILEDATA : L_MC1P_ProfileData;
END_VAR
END_METHOD

METHOD CALCPROFILE_40B4 : BOOL
VAR_INPUT
	LRSTARTACC : LREAL;
	LRSTARTVEL : LREAL;
	LRMAXACC : LREAL;
	LRMAXDEC : LREAL;
	LRMAXVEL : LREAL;
	LRTARGETACC : LREAL;
	LRTARGETVEL : LREAL;
	LRTARGETPOS : LREAL;
	LRJERKACC : LREAL;
	LRJERKDEC : LREAL;
	LRJERKTIMEACC : LREAL;
	LRJERKTIMEDEC : LREAL;
	SCMAXPROFILEDATA : L_MC1P_IntProfileData;
	SCMINPROFILEDATA : L_MC1P_IntProfileData;
END_VAR
VAR_OUTPUT
	DWSTATE : DWORD;
END_VAR
VAR_IN_OUT
	SCPROFILEDATA : L_MC1P_ProfileData;
	SCPROFILEPARAMETER : L_MC1P_ProfileParameter;
END_VAR
END_METHOD

METHOD CALCPROFILE_40B4_CALC : BOOL
VAR_INPUT
	LRSTARTACC : LREAL;
	LRSTARTVEL : LREAL;
	LRMAXACC : LREAL;
	LRMAXDEC : LREAL;
	LRMAXVEL : LREAL;
	LRTARGETACC : LREAL;
	LRTARGETVEL : LREAL;
	LRTARGETPOS : LREAL;
	LRJERKACC : LREAL;
	LRJERKDEC : LREAL;
	LRJERKTIMEACC : LREAL;
	LRJERKTIMEDEC : LREAL;
	T7 : LREAL;
END_VAR
VAR_IN_OUT
	SCPROFILEDATA : L_MC1P_ProfileData;
END_VAR
END_METHOD

METHOD CALCPROFILE_40B4_SEARCHTIMES : BOOL
VAR_INPUT
	LRSTARTACC : LREAL;
	LRSTARTVEL : LREAL;
	LRMAXACC : LREAL;
	LRMAXDEC : LREAL;
	LRMAXVEL : LREAL;
	LRTARGETACC : LREAL;
	LRTARGETVEL : LREAL;
	LRTARGETPOS : LREAL;
	LRJERKACC : LREAL;
	LRJERKDEC : LREAL;
	LRJERKTIMEACC : LREAL;
	LRJERKTIMEDEC : LREAL;
	T7_STARTVALUE : LREAL;
END_VAR
VAR_IN_OUT
	T7 : LREAL;
END_VAR
END_METHOD

METHOD CALCPROFILE_40BA : BOOL
VAR_INPUT
	LRSTARTACC : LREAL;
	LRSTARTVEL : LREAL;
	LRMAXACC : LREAL;
	LRMAXDEC : LREAL;
	LRMAXVEL : LREAL;
	LRTARGETACC : LREAL;
	LRTARGETVEL : LREAL;
	LRTARGETPOS : LREAL;
	LRJERKACC : LREAL;
	LRJERKDEC : LREAL;
	LRJERKTIMEACC : LREAL;
	LRJERKTIMEDEC : LREAL;
	SCMAXPROFILEDATA : L_MC1P_IntProfileData;
	SCMINPROFILEDATA : L_MC1P_IntProfileData;
END_VAR
VAR_OUTPUT
	DWSTATE : DWORD;
END_VAR
VAR_IN_OUT
	SCPROFILEDATA : L_MC1P_ProfileData;
	SCPROFILEPARAMETER : L_MC1P_ProfileParameter;
END_VAR
END_METHOD

METHOD CALCPROFILE_40BA_LINVELPH13_AEGE0 : BOOL
VAR_INPUT
	LRSTARTACC : LREAL;
	LRSTARTVEL : LREAL;
	LRMAXACC : LREAL;
	LRMAXDEC : LREAL;
	LRMAXVEL : LREAL;
	LRTARGETACC : LREAL;
	LRTARGETPOS : LREAL;
	LRJERKACC : LREAL;
	LRJERKDEC : LREAL;
	LRJERKTIMEACC : LREAL;
	LRJERKTIMEDEC : LREAL;
END_VAR
VAR_IN_OUT
	SCPROFILEDATA : L_MC1P_ProfileData;
END_VAR
END_METHOD

METHOD CALCPROFILE_40BA_LINVELPH13_AELT0 : BOOL
VAR_INPUT
	LRSTARTACC : LREAL;
	LRSTARTVEL : LREAL;
	LRMAXACC : LREAL;
	LRMAXDEC : LREAL;
	LRMAXVEL : LREAL;
	LRTARGETACC : LREAL;
	LRTARGETPOS : LREAL;
	LRJERKACC : LREAL;
	LRJERKDEC : LREAL;
	LRJERKTIMEACC : LREAL;
	LRJERKTIMEDEC : LREAL;
END_VAR
VAR_IN_OUT
	SCPROFILEDATA : L_MC1P_ProfileData;
END_VAR
END_METHOD

METHOD CALCPROFILE_40BA_LINVELPH17 : BOOL
VAR_INPUT
	LRSTARTACC : LREAL;
	LRSTARTVEL : LREAL;
	LRMAXACC : LREAL;
	LRMAXDEC : LREAL;
	LRMAXVEL : LREAL;
	LRTARGETACC : LREAL;
	LRTARGETPOS : LREAL;
END_VAR
VAR_IN_OUT
	SCPROFILEDATA : L_MC1P_ProfileData;
END_VAR
END_METHOD

METHOD CALCPROFILE_40BA_LINVELPH57 : BOOL
VAR_INPUT
	LRSTARTACC : LREAL;
	LRSTARTVEL : LREAL;
	LRMAXACC : LREAL;
	LRMAXDEC : LREAL;
	LRMAXVEL : LREAL;
	LRTARGETACC : LREAL;
	LRTARGETPOS : LREAL;
	LRJERKACC : LREAL;
	LRJERKDEC : LREAL;
	LRJERKTIMEACC : LREAL;
	LRJERKTIMEDEC : LREAL;
END_VAR
VAR_IN_OUT
	SCPROFILEDATA : L_MC1P_ProfileData;
END_VAR
END_METHOD

METHOD CALCPROFILE_40BA_A0LETAMAX_AEGE0 : BOOL
VAR_INPUT
	LRSTARTACC : LREAL;
	LRSTARTVEL : LREAL;
	LRMAXACC : LREAL;
	LRMAXDEC : LREAL;
	LRMAXVEL : LREAL;
	LRTARGETACC : LREAL;
	LRTARGETPOS : LREAL;
	LRJERKACC : LREAL;
	LRJERKDEC : LREAL;
	LRJERKTIMEACC : LREAL;
	LRJERKTIMEDEC : LREAL;
END_VAR
VAR_IN_OUT
	SCPROFILEDATA : L_MC1P_ProfileData;
END_VAR
END_METHOD

METHOD CALCPROFILE_40BA_A0LETAMAX_AELT0 : BOOL
VAR_INPUT
	LRSTARTACC : LREAL;
	LRSTARTVEL : LREAL;
	LRMAXACC : LREAL;
	LRMAXDEC : LREAL;
	LRMAXVEL : LREAL;
	LRTARGETACC : LREAL;
	LRTARGETPOS : LREAL;
	LRJERKACC : LREAL;
	LRJERKDEC : LREAL;
	LRJERKTIMEACC : LREAL;
	LRJERKTIMEDEC : LREAL;
END_VAR
VAR_IN_OUT
	SCPROFILEDATA : L_MC1P_ProfileData;
END_VAR
END_METHOD

METHOD CALCPROFILE_40C0 : BOOL
VAR_INPUT
	LRSTARTACC : LREAL;
	LRSTARTVEL : LREAL;
	LRMAXACC : LREAL;
	LRMAXDEC : LREAL;
	LRMAXVEL : LREAL;
	LRTARGETACC : LREAL;
	LRTARGETVEL : LREAL;
	LRTARGETPOS : LREAL;
	LRJERKACC : LREAL;
	LRJERKDEC : LREAL;
	LRJERKTIMEACC : LREAL;
	LRJERKTIMEDEC : LREAL;
	SCMAXPROFILEDATA : L_MC1P_IntProfileData;
	SCMINPROFILEDATA : L_MC1P_IntProfileData;
END_VAR
VAR_OUTPUT
	DWSTATE : DWORD;
END_VAR
VAR_IN_OUT
	SCPROFILEDATA : L_MC1P_ProfileData;
	SCPROFILEPARAMETER : L_MC1P_ProfileParameter;
END_VAR
END_METHOD

METHOD CALCPROFILE_40C0_LINVELPH57 : BOOL
VAR_INPUT
	LRSTARTACC : LREAL;
	LRSTARTVEL : LREAL;
	LRMAXACC : LREAL;
	LRMAXDEC : LREAL;
	LRMAXVEL : LREAL;
	LRTARGETACC : LREAL;
	LRTARGETVEL : LREAL;
	LRTARGETPOS : LREAL;
	LRJERKACC : LREAL;
	LRJERKDEC : LREAL;
	LRJERKTIMEACC : LREAL;
	LRJERKTIMEDEC : LREAL;
	T5 : LREAL;
	T7 : LREAL;
END_VAR
VAR_IN_OUT
	SCPROFILEDATA : L_MC1P_ProfileData;
END_VAR
END_METHOD

METHOD CALCPROFILE_40C0_LINVELPH57_SEARCHTIMEST5T7 : BOOL
VAR_INPUT
	LRSTARTACC : LREAL;
	LRSTARTVEL : LREAL;
	LRMAXACC : LREAL;
	LRMAXDEC : LREAL;
	LRMAXVEL : LREAL;
	LRTARGETACC : LREAL;
	LRTARGETVEL : LREAL;
	LRTARGETPOS : LREAL;
	LRMINPOSUNIT : LREAL;
	LRJERKACC : LREAL;
	LRJERKDEC : LREAL;
	LRJERKTIMEACC : LREAL;
	LRJERKTIMEDEC : LREAL;
	T5_STARTVALUE : LREAL;
	T7_STARTVALUE : LREAL;
END_VAR
VAR_IN_OUT
	T5 : LREAL;
	T7 : LREAL;
END_VAR
END_METHOD

METHOD CALCPROFILE_40C0_SEARCHTIMEST5T7 : BOOL
VAR_INPUT
	LRSTARTACC : LREAL;
	LRSTARTVEL : LREAL;
	LRMAXACC : LREAL;
	LRMAXDEC : LREAL;
	LRMAXVEL : LREAL;
	LRTARGETACC : LREAL;
	LRTARGETVEL : LREAL;
	LRTARGETPOS : LREAL;
	LRMINPOSUNIT : LREAL;
	LRJERKACC : LREAL;
	LRJERKDEC : LREAL;
	LRJERKTIMEACC : LREAL;
	LRJERKTIMEDEC : LREAL;
	T5_STARTVALUE : LREAL;
	T7_STARTVALUE : LREAL;
END_VAR
VAR_IN_OUT
	T5 : LREAL;
	T7 : LREAL;
END_VAR
END_METHOD

METHOD CALCPROFILE_40C0_A0LTAMAXT31 : BOOL
VAR_INPUT
	LRSTARTACC : LREAL;
	LRSTARTVEL : LREAL;
	LRMAXACC : LREAL;
	LRMAXDEC : LREAL;
	LRTARGETVEL : LREAL;
	LRTARGETPOS : LREAL;
	LRJERKACC : LREAL;
	LRJERKDEC : LREAL;
	LRJERKTIMEACC : LREAL;
	LRJERKTIMEDEC : LREAL;
END_VAR
VAR_IN_OUT
	SCPROFILEDATA : L_MC1P_ProfileData;
END_VAR
END_METHOD

METHOD CALCPROFILE_40C0_AELTAMAXT5T7 : BOOL
VAR_INPUT
	LRSTARTACC : LREAL;
	LRSTARTVEL : LREAL;
	LRMAXACC : LREAL;
	LRMAXDEC : LREAL;
	LRMAXVEL : LREAL;
	LRTARGETACC : LREAL;
	LRTARGETVEL : LREAL;
	LRTARGETPOS : LREAL;
	LRJERKACC : LREAL;
	LRJERKDEC : LREAL;
	LRJERKTIMEACC : LREAL;
	LRJERKTIMEDEC : LREAL;
	T5 : LREAL;
	T7 : LREAL;
END_VAR
VAR_IN_OUT
	SCPROFILEDATA : L_MC1P_ProfileData;
END_VAR
END_METHOD

METHOD CALCPROFILE_40CB : BOOL
VAR_INPUT
	LRSTARTACC : LREAL;
	LRSTARTVEL : LREAL;
	LRMAXACC : LREAL;
	LRMAXDEC : LREAL;
	LRMAXVEL : LREAL;
	LRTARGETACC : LREAL;
	LRTARGETVEL : LREAL;
	LRTARGETPOS : LREAL;
	LRJERKACC : LREAL;
	LRJERKDEC : LREAL;
	LRJERKTIMEACC : LREAL;
	LRJERKTIMEDEC : LREAL;
	SCMAXPROFILEDATA : L_MC1P_IntProfileData;
	SCMINPROFILEDATA : L_MC1P_IntProfileData;
END_VAR
VAR_OUTPUT
	DWSTATE : DWORD;
END_VAR
VAR_IN_OUT
	SCPROFILEDATA : L_MC1P_ProfileData;
	SCPROFILEPARAMETER : L_MC1P_ProfileParameter;
END_VAR
END_METHOD

METHOD CALCPROFILE_40CB_LINVELPH57 : BOOL
VAR_INPUT
	LRSTARTACC : LREAL;
	LRSTARTVEL : LREAL;
	LRMAXACC : LREAL;
	LRMAXDEC : LREAL;
	LRMAXVEL : LREAL;
	LRTARGETACC : LREAL;
	LRTARGETVEL : LREAL;
	LRTARGETPOS : LREAL;
	LRJERKACC : LREAL;
	LRJERKDEC : LREAL;
	LRJERKTIMEACC : LREAL;
	LRJERKTIMEDEC : LREAL;
	T7 : LREAL;
END_VAR
VAR_IN_OUT
	SCPROFILEDATA : L_MC1P_ProfileData;
END_VAR
END_METHOD

METHOD CALCPROFILE_40CB_LINVELPH57_SEARCHTIMES : BOOL
VAR_INPUT
	LRSTARTACC : LREAL;
	LRSTARTVEL : LREAL;
	LRMAXACC : LREAL;
	LRMAXDEC : LREAL;
	LRMAXVEL : LREAL;
	LRTARGETACC : LREAL;
	LRTARGETVEL : LREAL;
	LRTARGETPOS : LREAL;
	LRJERKACC : LREAL;
	LRJERKDEC : LREAL;
	LRJERKTIMEACC : LREAL;
	LRJERKTIMEDEC : LREAL;
	T7_MINVALUE : LREAL;
	T7_MAXVALUE : LREAL;
END_VAR
VAR_IN_OUT
	T7 : LREAL;
END_VAR
END_METHOD

METHOD CALCPROFILE_40CB_AOGET0 : BOOL
VAR_INPUT
	LRSTARTACC : LREAL;
	LRSTARTVEL : LREAL;
	LRMAXACC : LREAL;
	LRMAXDEC : LREAL;
	LRMAXVEL : LREAL;
	LRTARGETACC : LREAL;
	LRTARGETVEL : LREAL;
	LRTARGETPOS : LREAL;
	LRJERKACC : LREAL;
	LRJERKDEC : LREAL;
	LRJERKTIMEACC : LREAL;
	LRJERKTIMEDEC : LREAL;
	T7 : LREAL;
END_VAR
VAR_IN_OUT
	SCPROFILEDATA : L_MC1P_ProfileData;
END_VAR
END_METHOD

METHOD CALCPROFILE_40CBAOGET0_SEARCHTIMES : BOOL
VAR_INPUT
	LRSTARTACC : LREAL;
	LRSTARTVEL : LREAL;
	LRMAXACC : LREAL;
	LRMAXDEC : LREAL;
	LRMAXVEL : LREAL;
	LRTARGETACC : LREAL;
	LRTARGETVEL : LREAL;
	LRTARGETPOS : LREAL;
	LRJERKACC : LREAL;
	LRJERKDEC : LREAL;
	LRJERKTIMEACC : LREAL;
	LRJERKTIMEDEC : LREAL;
	T7_MINVALUE : LREAL;
	T7_MAXVALUE : LREAL;
END_VAR
VAR_IN_OUT
	T7 : LREAL;
END_VAR
END_METHOD

METHOD CALCPROFILE_40D0 : BOOL
VAR_INPUT
	LRSTARTACC : LREAL;
	LRSTARTVEL : LREAL;
	LRMAXACC : LREAL;
	LRMAXDEC : LREAL;
	LRMAXVEL : LREAL;
	LRTARGETACC : LREAL;
	LRTARGETVEL : LREAL;
	LRTARGETPOS : LREAL;
	LRJERKACC : LREAL;
	LRJERKDEC : LREAL;
	LRJERKTIMEACC : LREAL;
	LRJERKTIMEDEC : LREAL;
	SCMAXPROFILEDATA : L_MC1P_IntProfileData;
	SCMINPROFILEDATA : L_MC1P_IntProfileData;
END_VAR
VAR_OUTPUT
	DWSTATE : DWORD;
END_VAR
VAR_IN_OUT
	SCPROFILEDATA : L_MC1P_ProfileData;
	SCPROFILEPARAMETER : L_MC1P_ProfileParameter;
END_VAR
END_METHOD

METHOD CALCPROFILE_40D0_SEARCHTIMEST5T7 : BOOL
VAR_INPUT
	LRSTARTACC : LREAL;
	LRSTARTVEL : LREAL;
	LRMAXACC : LREAL;
	LRMAXDEC : LREAL;
	LRMAXVEL : LREAL;
	LRTARGETACC : LREAL;
	LRTARGETVEL : LREAL;
	LRTARGETPOS : LREAL;
	LRMINPOSUNIT : LREAL;
	LRJERKACC : LREAL;
	LRJERKDEC : LREAL;
	LRJERKTIMEACC : LREAL;
	LRJERKTIMEDEC : LREAL;
	T5_STARTVALUE : LREAL;
	T7_STARTVALUE : LREAL;
END_VAR
VAR_IN_OUT
	T5 : LREAL;
	T7 : LREAL;
END_VAR
END_METHOD

METHOD CALCPROFILE_40D0_A0LTAMAXT5T7 : BOOL
VAR_INPUT
	LRSTARTACC : LREAL;
	LRSTARTVEL : LREAL;
	LRMAXACC : LREAL;
	LRMAXDEC : LREAL;
	LRMAXVEL : LREAL;
	LRTARGETACC : LREAL;
	LRTARGETVEL : LREAL;
	LRTARGETPOS : LREAL;
	LRJERKACC : LREAL;
	LRJERKDEC : LREAL;
	LRJERKTIMEACC : LREAL;
	LRJERKTIMEDEC : LREAL;
	T5 : LREAL;
	T7 : LREAL;
END_VAR
VAR_IN_OUT
	SCPROFILEDATA : L_MC1P_ProfileData;
END_VAR
END_METHOD

METHOD CALCPROFILE_40D1 : BOOL
VAR_INPUT
	LRSTARTACC : LREAL;
	LRSTARTVEL : LREAL;
	LRMAXACC : LREAL;
	LRMAXDEC : LREAL;
	LRMAXVEL : LREAL;
	LRTARGETACC : LREAL;
	LRTARGETVEL : LREAL;
	LRTARGETPOS : LREAL;
	LRJERKACC : LREAL;
	LRJERKDEC : LREAL;
	LRJERKTIMEACC : LREAL;
	LRJERKTIMEDEC : LREAL;
	SCMAXPROFILEDATA : L_MC1P_IntProfileData;
	SCMINPROFILEDATA : L_MC1P_IntProfileData;
END_VAR
VAR_OUTPUT
	DWSTATE : DWORD;
END_VAR
VAR_IN_OUT
	SCPROFILEDATA : L_MC1P_ProfileData;
	SCPROFILEPARAMETER : L_MC1P_ProfileParameter;
END_VAR
END_METHOD

METHOD CALCPROFILE_40D1_AOGET0 : BOOL
VAR_INPUT
	LRSTARTACC : LREAL;
	LRSTARTVEL : LREAL;
	LRMAXACC : LREAL;
	LRMAXDEC : LREAL;
	LRMAXVEL : LREAL;
	LRTARGETACC : LREAL;
	LRTARGETVEL : LREAL;
	LRTARGETPOS : LREAL;
	LRJERKACC : LREAL;
	LRJERKDEC : LREAL;
	LRJERKTIMEACC : LREAL;
	LRJERKTIMEDEC : LREAL;
	T7 : LREAL;
END_VAR
VAR_IN_OUT
	SCPROFILEDATA : L_MC1P_ProfileData;
END_VAR
END_METHOD

METHOD CALCPROFILE_40D1_AOGET0_SEARCHTIMES : BOOL
VAR_INPUT
	LRSTARTACC : LREAL;
	LRSTARTVEL : LREAL;
	LRMAXACC : LREAL;
	LRMAXDEC : LREAL;
	LRMAXVEL : LREAL;
	LRTARGETACC : LREAL;
	LRTARGETVEL : LREAL;
	LRTARGETPOS : LREAL;
	LRMINPOSUNIT : LREAL;
	LRJERKACC : LREAL;
	LRJERKDEC : LREAL;
	LRJERKTIMEACC : LREAL;
	LRJERKTIMEDEC : LREAL;
	T7_STARTVALUE : LREAL;
END_VAR
VAR_IN_OUT
	T7 : LREAL;
END_VAR
END_METHOD

METHOD CALCPROFILE_40D1_AOLT0 : BOOL
VAR_INPUT
	LRSTARTACC : LREAL;
	LRSTARTVEL : LREAL;
	LRMAXACC : LREAL;
	LRMAXDEC : LREAL;
	LRMAXVEL : LREAL;
	LRTARGETACC : LREAL;
	LRTARGETVEL : LREAL;
	LRTARGETPOS : LREAL;
	LRJERKACC : LREAL;
	LRJERKDEC : LREAL;
	LRJERKTIMEACC : LREAL;
	LRJERKTIMEDEC : LREAL;
	T7 : LREAL;
END_VAR
VAR_IN_OUT
	SCPROFILEDATA : L_MC1P_ProfileData;
END_VAR
END_METHOD

METHOD CALCPROFILE_40D1_AOLT0_SEARCHTIMES : BOOL
VAR_INPUT
	LRSTARTACC : LREAL;
	LRSTARTVEL : LREAL;
	LRMAXACC : LREAL;
	LRMAXDEC : LREAL;
	LRMAXVEL : LREAL;
	LRTARGETACC : LREAL;
	LRTARGETVEL : LREAL;
	LRTARGETPOS : LREAL;
	LRMINPOSUNIT : LREAL;
	LRJERKACC : LREAL;
	LRJERKDEC : LREAL;
	LRJERKTIMEACC : LREAL;
	LRJERKTIMEDEC : LREAL;
	T7_STARTVALUE : LREAL;
END_VAR
VAR_IN_OUT
	T7 : LREAL;
END_VAR
END_METHOD

METHOD CALCPROFILE_40D2 : BOOL
VAR_INPUT
	LRSTARTACC : LREAL;
	LRSTARTVEL : LREAL;
	LRMAXACC : LREAL;
	LRMAXDEC : LREAL;
	LRMAXVEL : LREAL;
	LRTARGETACC : LREAL;
	LRTARGETVEL : LREAL;
	LRTARGETPOS : LREAL;
	LRJERKACC : LREAL;
	LRJERKDEC : LREAL;
	LRJERKTIMEACC : LREAL;
	LRJERKTIMEDEC : LREAL;
	SCMAXPROFILEDATA : L_MC1P_IntProfileData;
	SCMINPROFILEDATA : L_MC1P_IntProfileData;
END_VAR
VAR_OUTPUT
	DWSTATE : DWORD;
END_VAR
VAR_IN_OUT
	SCPROFILEDATA : L_MC1P_ProfileData;
	SCPROFILEPARAMETER : L_MC1P_ProfileParameter;
END_VAR
END_METHOD

METHOD CALCPROFILE_40D2_AOGE0_AEGT0
VAR_INPUT
	LRSTARTACC : LREAL;
	LRSTARTVEL : LREAL;
	LRMAXACC : LREAL;
	LRMAXDEC : LREAL;
	LRMAXVEL : LREAL;
	LRTARGETACC : LREAL;
	LRTARGETVEL : LREAL;
	LRTARGETPOS : LREAL;
	LRJERKACC : LREAL;
	LRJERKDEC : LREAL;
	LRJERKTIMEACC : LREAL;
	LRJERKTIMEDEC : LREAL;
	T7 : LREAL;
END_VAR
VAR_IN_OUT
	SCPROFILEDATA : L_MC1P_ProfileData;
END_VAR
END_METHOD

METHOD CALCPROFILE_40D2_AOGET0_AEGT0_SEARCHTIMES
VAR_INPUT
	LRSTARTACC : LREAL;
	LRSTARTVEL : LREAL;
	LRMAXACC : LREAL;
	LRMAXDEC : LREAL;
	LRMAXVEL : LREAL;
	LRTARGETACC : LREAL;
	LRTARGETVEL : LREAL;
	LRTARGETPOS : LREAL;
	LRJERKACC : LREAL;
	LRJERKDEC : LREAL;
	LRJERKTIMEACC : LREAL;
	LRJERKTIMEDEC : LREAL;
	T7_STARTVALUE : LREAL;
END_VAR
VAR_IN_OUT
	T7 : LREAL;
END_VAR
END_METHOD

METHOD CALCPROFILE_40D2_AOGET0_AELE0 : BOOL
VAR_INPUT
	LRSTARTACC : LREAL;
	LRSTARTVEL : LREAL;
	LRMAXACC : LREAL;
	LRMAXDEC : LREAL;
	LRMAXVEL : LREAL;
	LRTARGETACC : LREAL;
	LRTARGETVEL : LREAL;
	LRTARGETPOS : LREAL;
	LRJERKACC : LREAL;
	LRJERKDEC : LREAL;
	LRJERKTIMEACC : LREAL;
	LRJERKTIMEDEC : LREAL;
	T7 : LREAL;
END_VAR
VAR_IN_OUT
	SCPROFILEDATA : L_MC1P_ProfileData;
END_VAR
END_METHOD

METHOD CALCPROFILE_40D2_AOGET0_AELE0_SEARCHTIMES : BOOL
VAR_INPUT
	LRSTARTACC : LREAL;
	LRSTARTVEL : LREAL;
	LRMAXACC : LREAL;
	LRMAXDEC : LREAL;
	LRMAXVEL : LREAL;
	LRTARGETACC : LREAL;
	LRTARGETVEL : LREAL;
	LRTARGETPOS : LREAL;
	LRJERKACC : LREAL;
	LRJERKDEC : LREAL;
	LRJERKTIMEACC : LREAL;
	LRJERKTIMEDEC : LREAL;
	T7_STARTVALUE : LREAL;
END_VAR
VAR_IN_OUT
	T7 : LREAL;
END_VAR
END_METHOD

METHOD CALCPROFILE_40D2_AOLT0_AEGT0
VAR_INPUT
	LRSTARTACC : LREAL;
	LRSTARTVEL : LREAL;
	LRMAXACC : LREAL;
	LRMAXDEC : LREAL;
	LRMAXVEL : LREAL;
	LRTARGETACC : LREAL;
	LRTARGETVEL : LREAL;
	LRTARGETPOS : LREAL;
	LRJERKACC : LREAL;
	LRJERKDEC : LREAL;
	LRJERKTIMEACC : LREAL;
	LRJERKTIMEDEC : LREAL;
	T7 : LREAL;
END_VAR
VAR_IN_OUT
	SCPROFILEDATA : L_MC1P_ProfileData;
END_VAR
END_METHOD

METHOD CALCPROFILE_40D2_AOLT0_AEGT0_SEARCHTIMES
VAR_INPUT
	LRSTARTACC : LREAL;
	LRSTARTVEL : LREAL;
	LRMAXACC : LREAL;
	LRMAXDEC : LREAL;
	LRMAXVEL : LREAL;
	LRTARGETACC : LREAL;
	LRTARGETVEL : LREAL;
	LRTARGETPOS : LREAL;
	LRJERKACC : LREAL;
	LRJERKDEC : LREAL;
	LRJERKTIMEACC : LREAL;
	LRJERKTIMEDEC : LREAL;
	T7_STARTVALUE : LREAL;
END_VAR
VAR_IN_OUT
	T7 : LREAL;
END_VAR
END_METHOD

METHOD CALCPROFILE_40D2_AOLT0_AELE0 : BOOL
VAR_INPUT
	LRSTARTACC : LREAL;
	LRSTARTVEL : LREAL;
	LRMAXACC : LREAL;
	LRMAXDEC : LREAL;
	LRMAXVEL : LREAL;
	LRTARGETACC : LREAL;
	LRTARGETVEL : LREAL;
	LRTARGETPOS : LREAL;
	LRJERKACC : LREAL;
	LRJERKDEC : LREAL;
	LRJERKTIMEACC : LREAL;
	LRJERKTIMEDEC : LREAL;
	T7 : LREAL;
END_VAR
VAR_IN_OUT
	SCPROFILEDATA : L_MC1P_ProfileData;
END_VAR
END_METHOD

METHOD CALCPROFILE_40D2_AOLT0_AELE0_SEARCHTIMES : BOOL
VAR_INPUT
	LRSTARTACC : LREAL;
	LRSTARTVEL : LREAL;
	LRMAXACC : LREAL;
	LRMAXDEC : LREAL;
	LRMAXVEL : LREAL;
	LRTARGETACC : LREAL;
	LRTARGETVEL : LREAL;
	LRTARGETPOS : LREAL;
	LRJERKACC : LREAL;
	LRJERKDEC : LREAL;
	LRJERKTIMEACC : LREAL;
	LRJERKTIMEDEC : LREAL;
	T7_STARTVALUE : LREAL;
END_VAR
VAR_IN_OUT
	T7 : LREAL;
END_VAR
END_METHOD

METHOD CALCPROFILE_40D3 : BOOL
VAR_INPUT
	LRSTARTACC : LREAL;
	LRSTARTVEL : LREAL;
	LRMAXACC : LREAL;
	LRMAXDEC : LREAL;
	LRMAXVEL : LREAL;
	LRTARGETACC : LREAL;
	LRTARGETVEL : LREAL;
	LRTARGETPOS : LREAL;
	LRJERKACC : LREAL;
	LRJERKDEC : LREAL;
	LRJERKTIMEACC : LREAL;
	LRJERKTIMEDEC : LREAL;
	SCMAXPROFILEDATA : L_MC1P_IntProfileData;
	SCMINPROFILEDATA : L_MC1P_IntProfileData;
END_VAR
VAR_OUTPUT
	DWSTATE : DWORD;
END_VAR
VAR_IN_OUT
	SCPROFILEDATA : L_MC1P_ProfileData;
	SCPROFILEPARAMETER : L_MC1P_ProfileParameter;
END_VAR
END_METHOD

METHOD CALCPROFILE_40D3_CALC : BOOL
VAR_INPUT
	LRSTARTACC : LREAL;
	LRSTARTVEL : LREAL;
	LRMAXACC : LREAL;
	LRMAXDEC : LREAL;
	LRMAXVEL : LREAL;
	LRTARGETACC : LREAL;
	LRTARGETVEL : LREAL;
	LRTARGETPOS : LREAL;
	LRJERKACC : LREAL;
	LRJERKDEC : LREAL;
	LRJERKTIMEACC : LREAL;
	LRJERKTIMEDEC : LREAL;
	T7 : LREAL;
END_VAR
VAR_IN_OUT
	SCPROFILEDATA : L_MC1P_ProfileData;
END_VAR
END_METHOD

METHOD CALCPROFILE_40D3_SEARCHTIMES : BOOL
VAR_INPUT
	LRSTARTACC : LREAL;
	LRSTARTVEL : LREAL;
	LRMAXACC : LREAL;
	LRMAXDEC : LREAL;
	LRMAXVEL : LREAL;
	LRTARGETACC : LREAL;
	LRTARGETVEL : LREAL;
	LRTARGETPOS : LREAL;
	LRJERKACC : LREAL;
	LRJERKDEC : LREAL;
	LRJERKTIMEACC : LREAL;
	LRJERKTIMEDEC : LREAL;
	T7_STARTVALUE : LREAL;
END_VAR
VAR_IN_OUT
	T7 : LREAL;
END_VAR
END_METHOD

METHOD CALCPROFILE_40DA : BOOL
VAR_INPUT
	LRSTARTACC : LREAL;
	LRSTARTVEL : LREAL;
	LRMAXACC : LREAL;
	LRMAXDEC : LREAL;
	LRMAXVEL : LREAL;
	LRTARGETACC : LREAL;
	LRTARGETVEL : LREAL;
	LRTARGETPOS : LREAL;
	LRJERKACC : LREAL;
	LRJERKDEC : LREAL;
	LRJERKTIMEACC : LREAL;
	LRJERKTIMEDEC : LREAL;
	SCMAXPROFILEDATA : L_MC1P_IntProfileData;
	SCMINPROFILEDATA : L_MC1P_IntProfileData;
END_VAR
VAR_OUTPUT
	DWSTATE : DWORD;
END_VAR
VAR_IN_OUT
	SCPROFILEDATA : L_MC1P_ProfileData;
	SCPROFILEPARAMETER : L_MC1P_ProfileParameter;
END_VAR
END_METHOD

METHOD CALCPROFILE_40DA_AEGE0 : BOOL
VAR_INPUT
	LRSTARTACC : LREAL;
	LRSTARTVEL : LREAL;
	LRMAXACC : LREAL;
	LRMAXDEC : LREAL;
	LRMAXVEL : LREAL;
	LRTARGETACC : LREAL;
	LRTARGETVEL : LREAL;
	LRTARGETPOS : LREAL;
	LRJERKACC : LREAL;
	LRJERKDEC : LREAL;
	LRJERKTIMEACC : LREAL;
	LRJERKTIMEDEC : LREAL;
	T7 : LREAL;
END_VAR
VAR_IN_OUT
	SCPROFILEDATA : L_MC1P_ProfileData;
END_VAR
END_METHOD

METHOD CALCPROFILE_40DA_AELT0 : BOOL
VAR_INPUT
	LRSTARTACC : LREAL;
	LRSTARTVEL : LREAL;
	LRMAXACC : LREAL;
	LRMAXDEC : LREAL;
	LRMAXVEL : LREAL;
	LRTARGETACC : LREAL;
	LRTARGETVEL : LREAL;
	LRTARGETPOS : LREAL;
	LRJERKACC : LREAL;
	LRJERKDEC : LREAL;
	LRJERKTIMEACC : LREAL;
	LRJERKTIMEDEC : LREAL;
	T7 : LREAL;
END_VAR
VAR_IN_OUT
	SCPROFILEDATA : L_MC1P_ProfileData;
END_VAR
END_METHOD

METHOD CALCPROFILE_40DAAEGE0_SEARCHTIMES : BOOL
VAR_INPUT
	LRSTARTACC : LREAL;
	LRSTARTVEL : LREAL;
	LRMAXACC : LREAL;
	LRMAXDEC : LREAL;
	LRMAXVEL : LREAL;
	LRTARGETACC : LREAL;
	LRTARGETVEL : LREAL;
	LRTARGETPOS : LREAL;
	LRJERKACC : LREAL;
	LRJERKDEC : LREAL;
	LRJERKTIMEACC : LREAL;
	LRJERKTIMEDEC : LREAL;
	T7_MINVALUE : LREAL;
	T7_MAXVALUE : LREAL;
END_VAR
VAR_IN_OUT
	T7 : LREAL;
END_VAR
END_METHOD

METHOD CALCPROFILE_40DAAELT0_SEARCHTIMES : BOOL
VAR_INPUT
	LRSTARTACC : LREAL;
	LRSTARTVEL : LREAL;
	LRMAXACC : LREAL;
	LRMAXDEC : LREAL;
	LRMAXVEL : LREAL;
	LRTARGETACC : LREAL;
	LRTARGETVEL : LREAL;
	LRTARGETPOS : LREAL;
	LRJERKACC : LREAL;
	LRJERKDEC : LREAL;
	LRJERKTIMEACC : LREAL;
	LRJERKTIMEDEC : LREAL;
	T7_MINVALUE : LREAL;
	T7_MAXVALUE : LREAL;
END_VAR
VAR_OUTPUT
	T7 : LREAL;
END_VAR
END_METHOD

METHOD CALCPROFILE_40DB : BOOL
VAR_INPUT
	LRSTARTACC : LREAL;
	LRSTARTVEL : LREAL;
	LRMAXACC : LREAL;
	LRMAXDEC : LREAL;
	LRMAXVEL : LREAL;
	LRTARGETACC : LREAL;
	LRTARGETVEL : LREAL;
	LRTARGETPOS : LREAL;
	LRJERKACC : LREAL;
	LRJERKDEC : LREAL;
	LRJERKTIMEACC : LREAL;
	LRJERKTIMEDEC : LREAL;
	SCMAXPROFILEDATA : L_MC1P_IntProfileData;
	SCMINPROFILEDATA : L_MC1P_IntProfileData;
END_VAR
VAR_OUTPUT
	DWSTATE : DWORD;
END_VAR
VAR_IN_OUT
	SCPROFILEDATA : L_MC1P_ProfileData;
	SCPROFILEPARAMETER : L_MC1P_ProfileParameter;
END_VAR
END_METHOD

METHOD CALCPROFILE_40DB_AOGET0 : BOOL
VAR_INPUT
	LRSTARTACC : LREAL;
	LRSTARTVEL : LREAL;
	LRMAXACC : LREAL;
	LRMAXDEC : LREAL;
	LRMAXVEL : LREAL;
	LRTARGETACC : LREAL;
	LRTARGETVEL : LREAL;
	LRTARGETPOS : LREAL;
	LRJERKACC : LREAL;
	LRJERKDEC : LREAL;
	LRJERKTIMEACC : LREAL;
	LRJERKTIMEDEC : LREAL;
	T7 : LREAL;
END_VAR
VAR_IN_OUT
	SCPROFILEDATA : L_MC1P_ProfileData;
END_VAR
END_METHOD

METHOD CALCPROFILE_40DBAOGET0_SEARCHTIMES : BOOL
VAR_INPUT
	LRSTARTACC : LREAL;
	LRSTARTVEL : LREAL;
	LRMAXACC : LREAL;
	LRMAXDEC : LREAL;
	LRMAXVEL : LREAL;
	LRTARGETACC : LREAL;
	LRTARGETVEL : LREAL;
	LRTARGETPOS : LREAL;
	LRJERKACC : LREAL;
	LRJERKDEC : LREAL;
	LRJERKTIMEACC : LREAL;
	LRJERKTIMEDEC : LREAL;
	T7_MINVALUE : LREAL;
	T7_MAXVALUE : LREAL;
END_VAR
VAR_IN_OUT
	T7 : LREAL;
END_VAR
END_METHOD

METHOD CALCPROFILE_50A0 : BOOL
VAR_INPUT
	LRSTARTACC : LREAL;
	LRSTARTVEL : LREAL;
	LRMAXACC : LREAL;
	LRMAXDEC : LREAL;
	LRMAXVEL : LREAL;
	LRTARGETACC : LREAL;
	LRTARGETVEL : LREAL;
	LRTARGETPOS : LREAL;
	LRJERKACC : LREAL;
	LRJERKDEC : LREAL;
	LRJERKTIMEACC : LREAL;
	LRJERKTIMEDEC : LREAL;
	SCMAXPROFILEDATA : L_MC1P_IntProfileData;
	SCMINPROFILEDATA : L_MC1P_IntProfileData;
END_VAR
VAR_OUTPUT
	DWSTATE : DWORD;
END_VAR
VAR_IN_OUT
	SCPROFILEDATA : L_MC1P_ProfileData;
	SCPROFILEPARAMETER : L_MC1P_ProfileParameter;
END_VAR
END_METHOD

METHOD CALCPROFILE_50A0_A0GTAMAXT5T7 : BOOL
VAR_INPUT
	LRSTARTACC : LREAL;
	LRSTARTVEL : LREAL;
	LRMAXACC : LREAL;
	LRMAXDEC : LREAL;
	LRMAXVEL : LREAL;
	LRTARGETACC : LREAL;
	LRTARGETVEL : LREAL;
	LRTARGETPOS : LREAL;
	LRJERKACC : LREAL;
	LRJERKDEC : LREAL;
	LRJERKTIMEACC : LREAL;
	LRJERKTIMEDEC : LREAL;
	T5 : LREAL;
	T7 : LREAL;
END_VAR
VAR_IN_OUT
	SCPROFILEDATA : L_MC1P_ProfileData;
END_VAR
END_METHOD

METHOD CALCPROFILE_50A0_A0GTAMAX_SEARCHTIMEST5T7 : BOOL
VAR_INPUT
	LRSTARTACC : LREAL;
	LRSTARTVEL : LREAL;
	LRMAXACC : LREAL;
	LRMAXDEC : LREAL;
	LRMAXVEL : LREAL;
	LRTARGETACC : LREAL;
	LRTARGETVEL : LREAL;
	LRTARGETPOS : LREAL;
	LRMINPOSUNIT : LREAL;
	LRJERKACC : LREAL;
	LRJERKDEC : LREAL;
	LRJERKTIMEACC : LREAL;
	LRJERKTIMEDEC : LREAL;
	T5_STARTVALUE : LREAL;
	T7_STARTVALUE : LREAL;
END_VAR
VAR_IN_OUT
	T5 : LREAL;
	T7 : LREAL;
END_VAR
END_METHOD

METHOD CALCPROFILE_50B0 : BOOL
VAR_INPUT
	LRSTARTACC : LREAL;
	LRSTARTVEL : LREAL;
	LRMAXACC : LREAL;
	LRMAXDEC : LREAL;
	LRMAXVEL : LREAL;
	LRTARGETACC : LREAL;
	LRTARGETVEL : LREAL;
	LRTARGETPOS : LREAL;
	LRJERKACC : LREAL;
	LRJERKDEC : LREAL;
	LRJERKTIMEACC : LREAL;
	LRJERKTIMEDEC : LREAL;
	SCMAXPROFILEDATA : L_MC1P_IntProfileData;
	SCMINPROFILEDATA : L_MC1P_IntProfileData;
END_VAR
VAR_OUTPUT
	DWSTATE : DWORD;
END_VAR
VAR_IN_OUT
	SCPROFILEDATA : L_MC1P_ProfileData;
	SCPROFILEPARAMETER : L_MC1P_ProfileParameter;
END_VAR
END_METHOD

METHOD CALCPROFILE_50B0_A0GTAMAX_SEARCHTIMEST5T7 : BOOL
VAR_INPUT
	LRSTARTACC : LREAL;
	LRSTARTVEL : LREAL;
	LRMAXACC : LREAL;
	LRMAXDEC : LREAL;
	LRMAXVEL : LREAL;
	LRTARGETACC : LREAL;
	LRTARGETVEL : LREAL;
	LRTARGETPOS : LREAL;
	LRMINPOSUNIT : LREAL;
	LRJERKACC : LREAL;
	LRJERKDEC : LREAL;
	LRJERKTIMEACC : LREAL;
	LRJERKTIMEDEC : LREAL;
	T5_STARTVALUE : LREAL;
	T7_STARTVALUE : LREAL;
END_VAR
VAR_IN_OUT
	T5 : LREAL;
	T7 : LREAL;
END_VAR
END_METHOD

METHOD CALCPROFILE_50B0_A0GTAMAXT5T7 : BOOL
VAR_INPUT
	LRSTARTACC : LREAL;
	LRSTARTVEL : LREAL;
	LRMAXACC : LREAL;
	LRMAXDEC : LREAL;
	LRMAXVEL : LREAL;
	LRTARGETACC : LREAL;
	LRTARGETVEL : LREAL;
	LRTARGETPOS : LREAL;
	LRJERKACC : LREAL;
	LRJERKDEC : LREAL;
	LRJERKTIMEACC : LREAL;
	LRJERKTIMEDEC : LREAL;
	T5 : LREAL;
	T7 : LREAL;
END_VAR
VAR_IN_OUT
	SCPROFILEDATA : L_MC1P_ProfileData;
END_VAR
END_METHOD

METHOD CALCPROFILE_50B0_A0LTAMAXT5T7 : BOOL
VAR_INPUT
	LRSTARTACC : LREAL;
	LRSTARTVEL : LREAL;
	LRMAXACC : LREAL;
	LRMAXDEC : LREAL;
	LRMAXVEL : LREAL;
	LRTARGETACC : LREAL;
	LRTARGETVEL : LREAL;
	LRTARGETPOS : LREAL;
	LRJERKACC : LREAL;
	LRJERKDEC : LREAL;
	LRJERKTIMEACC : LREAL;
	LRJERKTIMEDEC : LREAL;
	T5 : LREAL;
	T7 : LREAL;
END_VAR
VAR_IN_OUT
	SCPROFILEDATA : L_MC1P_ProfileData;
END_VAR
END_METHOD

METHOD CALCPROFILE_50B0_A0LTAMAX_SEARCHTIMEST5T7 : BOOL
VAR_INPUT
	LRSTARTACC : LREAL;
	LRSTARTVEL : LREAL;
	LRMAXACC : LREAL;
	LRMAXDEC : LREAL;
	LRMAXVEL : LREAL;
	LRTARGETACC : LREAL;
	LRTARGETVEL : LREAL;
	LRTARGETPOS : LREAL;
	LRMINPOSUNIT : LREAL;
	LRJERKACC : LREAL;
	LRJERKDEC : LREAL;
	LRJERKTIMEACC : LREAL;
	LRJERKTIMEDEC : LREAL;
	T5_STARTVALUE : LREAL;
	T7_STARTVALUE : LREAL;
END_VAR
VAR_IN_OUT
	T5 : LREAL;
	T7 : LREAL;
END_VAR
END_METHOD

METHOD CALCPROFILE_50C0 : BOOL
VAR_INPUT
	LRSTARTACC : LREAL;
	LRSTARTVEL : LREAL;
	LRMAXACC : LREAL;
	LRMAXDEC : LREAL;
	LRMAXVEL : LREAL;
	LRTARGETACC : LREAL;
	LRTARGETVEL : LREAL;
	LRTARGETPOS : LREAL;
	LRJERKACC : LREAL;
	LRJERKDEC : LREAL;
	LRJERKTIMEACC : LREAL;
	LRJERKTIMEDEC : LREAL;
	SCMAXPROFILEDATA : L_MC1P_IntProfileData;
	SCMINPROFILEDATA : L_MC1P_IntProfileData;
END_VAR
VAR_OUTPUT
	DWSTATE : DWORD;
END_VAR
VAR_IN_OUT
	SCPROFILEDATA : L_MC1P_ProfileData;
	SCPROFILEPARAMETER : L_MC1P_ProfileParameter;
END_VAR
END_METHOD

METHOD CALCPROFILE_50C0_SEARCHTIMEST5T7 : BOOL
VAR_INPUT
	LRSTARTACC : LREAL;
	LRSTARTVEL : LREAL;
	LRMAXACC : LREAL;
	LRMAXDEC : LREAL;
	LRMAXVEL : LREAL;
	LRTARGETACC : LREAL;
	LRTARGETVEL : LREAL;
	LRTARGETPOS : LREAL;
	LRMINPOSUNIT : LREAL;
	LRJERKACC : LREAL;
	LRJERKDEC : LREAL;
	LRJERKTIMEACC : LREAL;
	LRJERKTIMEDEC : LREAL;
	T5_STARTVALUE : LREAL;
	T7_STARTVALUE : LREAL;
END_VAR
VAR_IN_OUT
	T5 : LREAL;
	T7 : LREAL;
END_VAR
END_METHOD

METHOD CALCPROFILE_50C0_A0LTAMAXT5T7 : BOOL
VAR_INPUT
	LRSTARTACC : LREAL;
	LRSTARTVEL : LREAL;
	LRMAXACC : LREAL;
	LRMAXDEC : LREAL;
	LRMAXVEL : LREAL;
	LRTARGETACC : LREAL;
	LRTARGETVEL : LREAL;
	LRTARGETPOS : LREAL;
	LRJERKACC : LREAL;
	LRJERKDEC : LREAL;
	LRJERKTIMEACC : LREAL;
	LRJERKTIMEDEC : LREAL;
	T5 : LREAL;
	T7 : LREAL;
END_VAR
VAR_IN_OUT
	SCPROFILEDATA : L_MC1P_ProfileData;
END_VAR
END_METHOD

METHOD CALCPROFILE_50D0 : BOOL
VAR_INPUT
	LRSTARTACC : LREAL;
	LRSTARTVEL : LREAL;
	LRMAXACC : LREAL;
	LRMAXDEC : LREAL;
	LRMAXVEL : LREAL;
	LRTARGETACC : LREAL;
	LRTARGETVEL : LREAL;
	LRTARGETPOS : LREAL;
	LRJERKACC : LREAL;
	LRJERKDEC : LREAL;
	LRJERKTIMEACC : LREAL;
	LRJERKTIMEDEC : LREAL;
	SCMAXPROFILEDATA : L_MC1P_IntProfileData;
	SCMINPROFILEDATA : L_MC1P_IntProfileData;
END_VAR
VAR_OUTPUT
	DWSTATE : DWORD;
END_VAR
VAR_IN_OUT
	SCPROFILEDATA : L_MC1P_ProfileData;
	SCPROFILEPARAMETER : L_MC1P_ProfileParameter;
END_VAR
END_METHOD

METHOD CALCPROFILE_50D0_SEARCHTIMEST5T7 : BOOL
VAR_INPUT
	LRSTARTACC : LREAL;
	LRSTARTVEL : LREAL;
	LRMAXACC : LREAL;
	LRMAXDEC : LREAL;
	LRMAXVEL : LREAL;
	LRTARGETACC : LREAL;
	LRTARGETVEL : LREAL;
	LRTARGETPOS : LREAL;
	LRMINPOSUNIT : LREAL;
	LRJERKACC : LREAL;
	LRJERKDEC : LREAL;
	LRJERKTIMEACC : LREAL;
	LRJERKTIMEDEC : LREAL;
	T5_STARTVALUE : LREAL;
	T7_STARTVALUE : LREAL;
END_VAR
VAR_IN_OUT
	T5 : LREAL;
	T7 : LREAL;
END_VAR
END_METHOD

METHOD CALCPROFILE_50D0_A0LTAMAXT5T7 : BOOL
VAR_INPUT
	LRSTARTACC : LREAL;
	LRSTARTVEL : LREAL;
	LRMAXACC : LREAL;
	LRMAXDEC : LREAL;
	LRMAXVEL : LREAL;
	LRTARGETACC : LREAL;
	LRTARGETVEL : LREAL;
	LRTARGETPOS : LREAL;
	LRJERKACC : LREAL;
	LRJERKDEC : LREAL;
	LRJERKTIMEACC : LREAL;
	LRJERKTIMEDEC : LREAL;
	T5 : LREAL;
	T7 : LREAL;
END_VAR
VAR_IN_OUT
	SCPROFILEDATA : L_MC1P_ProfileData;
END_VAR
END_METHOD

METHOD CALCPROFILE_50E0 : BOOL
VAR_INPUT
	LRSTARTACC : LREAL;
	LRSTARTVEL : LREAL;
	LRMAXACC : LREAL;
	LRMAXDEC : LREAL;
	LRMAXVEL : LREAL;
	LRTARGETACC : LREAL;
	LRTARGETVEL : LREAL;
	LRTARGETPOS : LREAL;
	LRJERKACC : LREAL;
	LRJERKDEC : LREAL;
	LRJERKTIMEACC : LREAL;
	LRJERKTIMEDEC : LREAL;
	SCMAXPROFILEDATA : L_MC1P_IntProfileData;
	SCMINPROFILEDATA : L_MC1P_IntProfileData;
END_VAR
VAR_OUTPUT
	DWSTATE : DWORD;
END_VAR
VAR_IN_OUT
	SCPROFILEDATA : L_MC1P_ProfileData;
	SCPROFILEPARAMETER : L_MC1P_ProfileParameter;
END_VAR
END_METHOD

METHOD CALCPROFILE_50E0_PROFILEDATA : BOOL
VAR_INPUT
	LRSTARTACC : LREAL;
	LRSTARTVEL : LREAL;
	LRMAXACC : LREAL;
	LRMAXDEC : LREAL;
	LRMAXVEL : LREAL;
	LRTARGETACC : LREAL;
	LRTARGETVEL : LREAL;
	LRTARGETPOS : LREAL;
	LRJERKACC : LREAL;
	LRJERKDEC : LREAL;
	LRJERKTIMEACC : LREAL;
	LRJERKTIMEDEC : LREAL;
	T5 : LREAL;
	T7 : LREAL;
END_VAR
VAR_IN_OUT
	SCPROFILEDATA : L_MC1P_ProfileData;
END_VAR
END_METHOD

METHOD CALCPROFILE_50E0_SEARCHTIMEST5T7 : BOOL
VAR_INPUT
	LRSTARTACC : LREAL;
	LRSTARTVEL : LREAL;
	LRMAXACC : LREAL;
	LRMAXDEC : LREAL;
	LRMAXVEL : LREAL;
	LRTARGETACC : LREAL;
	LRTARGETVEL : LREAL;
	LRTARGETPOS : LREAL;
	LRMINPOSUNIT : LREAL;
	LRJERKACC : LREAL;
	LRJERKDEC : LREAL;
	LRJERKTIMEACC : LREAL;
	LRJERKTIMEDEC : LREAL;
	T5_STARTVALUE : LREAL;
	T7_STARTVALUE : LREAL;
END_VAR
VAR_IN_OUT
	T5 : LREAL;
	T7 : LREAL;
END_VAR
END_METHOD

METHOD CALCPROFILE_50F0 : BOOL
VAR_INPUT
	LRSTARTACC : LREAL;
	LRSTARTVEL : LREAL;
	LRMAXACC : LREAL;
	LRMAXDEC : LREAL;
	LRMAXVEL : LREAL;
	LRTARGETACC : LREAL;
	LRTARGETVEL : LREAL;
	LRTARGETPOS : LREAL;
	LRJERKACC : LREAL;
	LRJERKDEC : LREAL;
	LRJERKTIMEACC : LREAL;
	LRJERKTIMEDEC : LREAL;
	SCMAXPROFILEDATA : L_MC1P_IntProfileData;
	SCMINPROFILEDATA : L_MC1P_IntProfileData;
END_VAR
VAR_OUTPUT
	DWSTATE : DWORD;
END_VAR
VAR_IN_OUT
	SCPROFILEDATA : L_MC1P_ProfileData;
	SCPROFILEPARAMETER : L_MC1P_ProfileParameter;
END_VAR
END_METHOD

METHOD CALCPROFILE_50F0_PROFILEDATA : BOOL
VAR_INPUT
	LRSTARTACC : LREAL;
	LRSTARTVEL : LREAL;
	LRMAXACC : LREAL;
	LRMAXDEC : LREAL;
	LRMAXVEL : LREAL;
	LRTARGETACC : LREAL;
	LRTARGETVEL : LREAL;
	LRTARGETPOS : LREAL;
	LRJERKACC : LREAL;
	LRJERKDEC : LREAL;
	LRJERKTIMEACC : LREAL;
	LRJERKTIMEDEC : LREAL;
	T5 : LREAL;
	T7 : LREAL;
END_VAR
VAR_IN_OUT
	SCPROFILEDATA : L_MC1P_ProfileData;
END_VAR
END_METHOD

METHOD CALCPROFILE_50F0_SEARCHTIMEST5T7 : BOOL
VAR_INPUT
	LRSTARTACC : LREAL;
	LRSTARTVEL : LREAL;
	LRMAXACC : LREAL;
	LRMAXDEC : LREAL;
	LRMAXVEL : LREAL;
	LRTARGETACC : LREAL;
	LRTARGETVEL : LREAL;
	LRTARGETPOS : LREAL;
	LRMINPOSUNIT : LREAL;
	LRJERKACC : LREAL;
	LRJERKDEC : LREAL;
	LRJERKTIMEACC : LREAL;
	LRJERKTIMEDEC : LREAL;
	T5_STARTVALUE : LREAL;
	T7_STARTVALUE : LREAL;
END_VAR
VAR_IN_OUT
	T5 : LREAL;
	T7 : LREAL;
END_VAR
END_METHOD

METHOD CALCPROFILE_60C0 : BOOL
VAR_INPUT
	LRSTARTACC : LREAL;
	LRSTARTVEL : LREAL;
	LRMAXACC : LREAL;
	LRMAXDEC : LREAL;
	LRMAXVEL : LREAL;
	LRTARGETACC : LREAL;
	LRTARGETVEL : LREAL;
	LRTARGETPOS : LREAL;
	LRJERKDEC : LREAL;
	SCMAXPROFILEDATA : L_MC1P_IntProfileData;
	SCMINPROFILEDATA : L_MC1P_IntProfileData;
END_VAR
VAR_OUTPUT
	DWSTATE : DWORD;
END_VAR
VAR_IN_OUT
	SCPROFILEDATA : L_MC1P_ProfileData;
	SCPROFILEPARAMETER : L_MC1P_ProfileParameter;
END_VAR
END_METHOD

METHOD CALCPROFILE_60C0_INCRJERKDEC : BOOL
VAR_INPUT
	LRSTARTACC : LREAL;
	LRSTARTVEL : LREAL;
	LRMAXACC : LREAL;
	LRMAXDEC : LREAL;
	LRMAXVEL : LREAL;
	LRTARGETACC : LREAL;
	LRTARGETVEL : LREAL;
	LRTARGETPOS : LREAL;
	J5 : LREAL;
END_VAR
VAR_OUTPUT
	DWSTATE : DWORD;
END_VAR
VAR_IN_OUT
	SCPROFILEDATA : L_MC1P_ProfileData;
END_VAR
END_METHOD

METHOD CALCPROFILE_60C0_SEARCHJERKDEC : BOOL
VAR_INPUT
	LRSTARTACC : LREAL;
	LRSTARTVEL : LREAL;
	LRMAXACC : LREAL;
	LRMAXDEC : LREAL;
	LRMAXVEL : LREAL;
	LRTARGETACC : LREAL;
	LRTARGETVEL : LREAL;
	LRTARGETPOS : LREAL;
	LRMINPOSUNIT : LREAL;
	J5_STARTVALUE : LREAL;
END_VAR
VAR_IN_OUT
	J5 : LREAL;
END_VAR
END_METHOD

METHOD CALCPROFILE_60D0 : BOOL
VAR_INPUT
	LRSTARTACC : LREAL;
	LRSTARTVEL : LREAL;
	LRMAXACC : LREAL;
	LRMAXDEC : LREAL;
	LRMAXVEL : LREAL;
	LRTARGETACC : LREAL;
	LRTARGETVEL : LREAL;
	LRTARGETPOS : LREAL;
	LRJERKDEC : LREAL;
	SCMAXPROFILEDATA : L_MC1P_IntProfileData;
	SCMINPROFILEDATA : L_MC1P_IntProfileData;
END_VAR
VAR_OUTPUT
	DWSTATE : DWORD;
END_VAR
VAR_IN_OUT
	SCPROFILEDATA : L_MC1P_ProfileData;
	SCPROFILEPARAMETER : L_MC1P_ProfileParameter;
END_VAR
END_METHOD

METHOD CALCPROFILE_60D0_INCRJERKDEC : BOOL
VAR_INPUT
	LRSTARTACC : LREAL;
	LRSTARTVEL : LREAL;
	LRMAXACC : LREAL;
	LRMAXDEC : LREAL;
	LRMAXVEL : LREAL;
	LRTARGETACC : LREAL;
	LRTARGETVEL : LREAL;
	LRTARGETPOS : LREAL;
	J5 : LREAL;
END_VAR
VAR_OUTPUT
	DWSTATE : DWORD;
END_VAR
VAR_IN_OUT
	SCPROFILEDATA : L_MC1P_ProfileData;
END_VAR
END_METHOD

METHOD CALCPROFILE_60D0_SEARCHJERKDEC : BOOL
VAR_INPUT
	LRSTARTACC : LREAL;
	LRSTARTVEL : LREAL;
	LRMAXACC : LREAL;
	LRMAXDEC : LREAL;
	LRMAXVEL : LREAL;
	LRTARGETACC : LREAL;
	LRTARGETVEL : LREAL;
	LRTARGETPOS : LREAL;
	LRMINPOSUNIT : LREAL;
	J5_STARTVALUE : LREAL;
END_VAR
VAR_IN_OUT
	J5 : LREAL;
END_VAR
END_METHOD

METHOD CALCPROFILE_6000 : BOOL
VAR_INPUT
	LRSTARTACC : LREAL;
	LRSTARTVEL : LREAL;
	LRMAXACC : LREAL;
	LRMAXDEC : LREAL;
	LRMAXVEL : LREAL;
	LRTARGETACC : LREAL;
	LRTARGETVEL : LREAL;
	LRTARGETPOS : LREAL;
	LRJERKACC : LREAL;
	LRJERKDEC : LREAL;
	LRJERKTIMEACC : LREAL;
	LRJERKTIMEDEC : LREAL;
	SCMINPROFILEDATA : L_MC1P_IntProfileData;
	SCMAXPROFILEDATA : L_MC1P_IntProfileData;
END_VAR
VAR_OUTPUT
	DWSTATE : DWORD;
END_VAR
VAR_IN_OUT
	SCPROFILEDATA : L_MC1P_ProfileData;
	SCPROFILEPARAMETER : L_MC1P_ProfileParameter;
END_VAR
END_METHOD

METHOD CALCPROFILE_6001 : BOOL
VAR_INPUT
	LRSTARTACC : LREAL;
	LRSTARTVEL : LREAL;
	LRMAXACC : LREAL;
	LRMAXDEC : LREAL;
	LRMAXVEL : LREAL;
	LRTARGETACC : LREAL;
	LRTARGETVEL : LREAL;
	LRTARGETPOS : LREAL;
	LRJERKACC : LREAL;
	LRJERKDEC : LREAL;
	LRJERKTIMEACC : LREAL;
	LRJERKTIMEDEC : LREAL;
	SCMINPROFILEDATA : L_MC1P_IntProfileData;
	SCMAXPROFILEDATA : L_MC1P_IntProfileData;
END_VAR
VAR_OUTPUT
	DWSTATE : DWORD;
END_VAR
VAR_IN_OUT
	SCPROFILEDATA : L_MC1P_ProfileData;
	SCPROFILEPARAMETER : L_MC1P_ProfileParameter;
END_VAR
END_METHOD

METHOD CALCPROFILE_6002 : BOOL
VAR_INPUT
	LRSTARTACC : LREAL;
	LRSTARTVEL : LREAL;
	LRMAXACC : LREAL;
	LRMAXDEC : LREAL;
	LRMAXVEL : LREAL;
	LRTARGETACC : LREAL;
	LRTARGETVEL : LREAL;
	LRTARGETPOS : LREAL;
	LRJERKACC : LREAL;
	LRJERKDEC : LREAL;
	LRJERKTIMEACC : LREAL;
	LRJERKTIMEDEC : LREAL;
	SCMINPROFILEDATA : L_MC1P_IntProfileData;
	SCMAXPROFILEDATA : L_MC1P_IntProfileData;
END_VAR
VAR_OUTPUT
	DWSTATE : DWORD;
END_VAR
VAR_IN_OUT
	SCPROFILEDATA : L_MC1P_ProfileData;
	SCPROFILEPARAMETER : L_MC1P_ProfileParameter;
END_VAR
END_METHOD

METHOD CALCPROFILE_6010 : BOOL
VAR_INPUT
	LRSTARTACC : LREAL;
	LRSTARTVEL : LREAL;
	LRMAXACC : LREAL;
	LRMAXDEC : LREAL;
	LRMAXVEL : LREAL;
	LRTARGETACC : LREAL;
	LRTARGETVEL : LREAL;
	LRTARGETPOS : LREAL;
	LRJERKACC : LREAL;
	LRJERKDEC : LREAL;
	LRJERKTIMEACC : LREAL;
	LRJERKTIMEDEC : LREAL;
	SCMINPROFILEDATA : L_MC1P_IntProfileData;
	SCMAXPROFILEDATA : L_MC1P_IntProfileData;
END_VAR
VAR_OUTPUT
	DWSTATE : DWORD;
END_VAR
VAR_IN_OUT
	SCPROFILEDATA : L_MC1P_ProfileData;
	SCPROFILEPARAMETER : L_MC1P_ProfileParameter;
END_VAR
END_METHOD

METHOD CALCPROFILE_60A0 : BOOL
VAR_INPUT
	LRSTARTACC : LREAL;
	LRSTARTVEL : LREAL;
	LRMAXACC : LREAL;
	LRMAXDEC : LREAL;
	LRMAXVEL : LREAL;
	LRTARGETACC : LREAL;
	LRTARGETVEL : LREAL;
	LRTARGETPOS : LREAL;
	LRJERKACC : LREAL;
	LRJERKDEC : LREAL;
	LRJERKTIMEACC : LREAL;
	LRJERKTIMEDEC : LREAL;
	SCMAXPROFILEDATA : L_MC1P_IntProfileData;
	SCMINPROFILEDATA : L_MC1P_IntProfileData;
END_VAR
VAR_OUTPUT
	DWSTATE : DWORD;
END_VAR
VAR_IN_OUT
	SCPROFILEDATA : L_MC1P_ProfileData;
	SCPROFILEPARAMETER : L_MC1P_ProfileParameter;
END_VAR
END_METHOD

METHOD CALCPROFILE_65E0 : BOOL
VAR_INPUT
	LRSTARTACC : LREAL;
	LRSTARTVEL : LREAL;
	LRMAXACC : LREAL;
	LRMAXDEC : LREAL;
	LRMAXVEL : LREAL;
	LRTARGETACC : LREAL;
	LRTARGETVEL : LREAL;
	LRTARGETPOS : LREAL;
	LRJERKACC : LREAL;
	LRJERKDEC : LREAL;
	LRJERKTIMEACC : LREAL;
	LRJERKTIMEDEC : LREAL;
	SCMINPROFILEDATA : L_MC1P_IntProfileData;
	SCMAXPROFILEDATA : L_MC1P_IntProfileData;
END_VAR
VAR_OUTPUT
	DWSTATE : DWORD;
END_VAR
VAR_IN_OUT
	SCPROFILEDATA : L_MC1P_ProfileData;
	SCPROFILEPARAMETER : L_MC1P_ProfileParameter;
END_VAR
END_METHOD

METHOD CALCPROFILE_65F0 : BOOL
VAR_INPUT
	LRSTARTACC : LREAL;
	LRSTARTVEL : LREAL;
	LRMAXACC : LREAL;
	LRMAXDEC : LREAL;
	LRMAXVEL : LREAL;
	LRTARGETACC : LREAL;
	LRTARGETVEL : LREAL;
	LRTARGETPOS : LREAL;
	LRJERKACC : LREAL;
	LRJERKDEC : LREAL;
	LRJERKTIMEACC : LREAL;
	LRJERKTIMEDEC : LREAL;
	SCMINPROFILEDATA : L_MC1P_IntProfileData;
	SCMAXPROFILEDATA : L_MC1P_IntProfileData;
END_VAR
VAR_OUTPUT
	DWSTATE : DWORD;
END_VAR
VAR_IN_OUT
	SCPROFILEDATA : L_MC1P_ProfileData;
	SCPROFILEPARAMETER : L_MC1P_ProfileParameter;
END_VAR
END_METHOD

METHOD CALCPROFILE_70E0 : BOOL
VAR_INPUT
	LRSTARTACC : LREAL;
	LRSTARTVEL : LREAL;
	LRMAXACC : LREAL;
	LRMAXDEC : LREAL;
	LRMAXVEL : LREAL;
	LRTARGETACC : LREAL;
	LRTARGETVEL : LREAL;
	LRTARGETPOS : LREAL;
	LRJERKACC : LREAL;
	LRJERKDEC : LREAL;
	LRJERKTIMEACC : LREAL;
	LRJERKTIMEDEC : LREAL;
	SCMAXPROFILEDATA : L_MC1P_IntProfileData;
	SCMINPROFILEDATA : L_MC1P_IntProfileData;
END_VAR
VAR_OUTPUT
	DWSTATE : DWORD;
END_VAR
VAR_IN_OUT
	SCPROFILEDATA : L_MC1P_ProfileData;
	SCPROFILEPARAMETER : L_MC1P_ProfileParameter;
END_VAR
END_METHOD

METHOD CALCPROFILE_70X0 : BOOL
VAR_INPUT
	LRSTARTACC : LREAL;
	LRSTARTVEL : LREAL;
	LRMAXACC : LREAL;
	LRMAXDEC : LREAL;
	LRMAXVEL : LREAL;
	LRTARGETACC : LREAL;
	LRTARGETVEL : LREAL;
	LRTARGETPOS : LREAL;
	LRJERKACC : LREAL;
	LRJERKDEC : LREAL;
	LRJERKTIMEACC : LREAL;
	LRJERKTIMEDEC : LREAL;
	SCMAXPROFILEDATA : L_MC1P_IntProfileData;
	SCMINPROFILEDATA : L_MC1P_IntProfileData;
END_VAR
VAR_OUTPUT
	DWSTATE : DWORD;
END_VAR
VAR_IN_OUT
	SCPROFILEDATA : L_MC1P_ProfileData;
	SCPROFILEPARAMETER : L_MC1P_ProfileParameter;
END_VAR
END_METHOD

METHOD CALCLINPROFILE_80B0
VAR_INPUT
	LRSTARTACC : LREAL;
	LRSTARTVEL : LREAL;
	SCPROFILEPARAMETER : L_MC1P_ProfileParameter;
	SCMINPROFILEDATA : L_MC1P_IntProfileData;
END_VAR
VAR_OUTPUT
	SCPROFILEDATA : L_MC1P_ProfileData;
END_VAR
END_METHOD

METHOD CALCPROFILE_80BA
VAR_INPUT
	LRSTARTACC : LREAL;
	LRSTARTVEL : LREAL;
	LRMAXACC : LREAL;
	LRMAXDEC : LREAL;
	LRMAXVEL : LREAL;
	LRTARGETACC : LREAL;
	LRTARGETVEL : LREAL;
	LRTARGETPOS : LREAL;
	LRJERKACC : LREAL;
	LRJERKDEC : LREAL;
	LRJERKTIMEACC : LREAL;
	LRJERKTIMEDEC : LREAL;
	SCMAXPROFILEDATA : L_MC1P_IntProfileData;
	SCMINPROFILEDATA : L_MC1P_IntProfileData;
END_VAR
VAR_OUTPUT
	DWSTATE : DWORD;
END_VAR
VAR_IN_OUT
	SCPROFILEDATA : L_MC1P_ProfileData;
	SCPROFILEPARAMETER : L_MC1P_ProfileParameter;
END_VAR
END_METHOD

METHOD CALCPROFILE_80BA_PROFILEDATA
VAR_INPUT
	LRSTARTACC : LREAL;
	LRSTARTVEL : LREAL;
	LRMAXACC : LREAL;
	LRMAXDEC : LREAL;
	LRMAXVEL : LREAL;
	LRTARGETACC : LREAL;
	LRTARGETVEL : LREAL;
	LRTARGETPOS : LREAL;
	LRJERKACC : LREAL;
	LRJERKDEC : LREAL;
	LRJERKTIMEACC : LREAL;
	LRJERKTIMEDEC : LREAL;
	T01 : LREAL;
	T12 : LREAL;
	T23 : LREAL;
	T5 : LREAL;
END_VAR
VAR_IN_OUT
	SCPROFILEDATA : L_MC1P_ProfileData;
END_VAR
END_METHOD

METHOD CALCPROFILE_80BB
VAR_INPUT
	LRSTARTACC : LREAL;
	LRSTARTVEL : LREAL;
	LRMAXACC : LREAL;
	LRMAXDEC : LREAL;
	LRMAXVEL : LREAL;
	LRTARGETACC : LREAL;
	LRTARGETVEL : LREAL;
	LRTARGETPOS : LREAL;
	LRJERKACC : LREAL;
	LRJERKDEC : LREAL;
	LRJERKTIMEACC : LREAL;
	LRJERKTIMEDEC : LREAL;
	SCMAXPROFILEDATA : L_MC1P_IntProfileData;
	SCMINPROFILEDATA : L_MC1P_IntProfileData;
END_VAR
VAR_OUTPUT
	DWSTATE : DWORD;
END_VAR
VAR_IN_OUT
	SCPROFILEDATA : L_MC1P_ProfileData;
	SCPROFILEPARAMETER : L_MC1P_ProfileParameter;
END_VAR
END_METHOD

METHOD CALCPROFILE_80BB_CALCT5
VAR_INPUT
	LRSTARTACC : LREAL;
	LRSTARTVEL : LREAL;
	LRMAXACC : LREAL;
	LRMAXDEC : LREAL;
	LRMAXVEL : LREAL;
	LRTARGETACC : LREAL;
	LRTARGETVEL : LREAL;
	LRTARGETPOS : LREAL;
	LRMINPOSUNIT : LREAL;
	LRJERKACC : LREAL;
	LRJERKDEC : LREAL;
	LRJERKTIMEACC : LREAL;
	LRJERKTIMEDEC : LREAL;
	T01 : LREAL;
	T12 : LREAL;
	T23 : LREAL;
END_VAR
VAR_OUTPUT
	T5 : ARRAY [1..2] OF LREAL;
END_VAR
END_METHOD

METHOD CALCPROFILE_80BB_PROFILEDATA
VAR_INPUT
	LRSTARTACC : LREAL;
	LRSTARTVEL : LREAL;
	LRMAXACC : LREAL;
	LRMAXDEC : LREAL;
	LRMAXVEL : LREAL;
	LRTARGETACC : LREAL;
	LRTARGETVEL : LREAL;
	LRTARGETPOS : LREAL;
	LRJERKACC : LREAL;
	LRJERKDEC : LREAL;
	LRJERKTIMEACC : LREAL;
	LRJERKTIMEDEC : LREAL;
	T01 : LREAL;
	T12 : LREAL;
	T23 : LREAL;
	T5 : LREAL;
END_VAR
VAR_IN_OUT
	SCPROFILEDATA : L_MC1P_ProfileData;
END_VAR
END_METHOD

METHOD CALCPROFILE_80BC
VAR_INPUT
	LRSTARTACC : LREAL;
	LRSTARTVEL : LREAL;
	LRMAXACC : LREAL;
	LRMAXDEC : LREAL;
	LRMAXVEL : LREAL;
	LRTARGETACC : LREAL;
	LRTARGETVEL : LREAL;
	LRTARGETPOS : LREAL;
	LRJERKACC : LREAL;
	LRJERKDEC : LREAL;
	LRJERKTIMEACC : LREAL;
	LRJERKTIMEDEC : LREAL;
	SCMAXPROFILEDATA : L_MC1P_IntProfileData;
	SCMINPROFILEDATA : L_MC1P_IntProfileData;
END_VAR
VAR_OUTPUT
	DWSTATE : DWORD;
END_VAR
VAR_IN_OUT
	SCPROFILEDATA : L_MC1P_ProfileData;
	SCPROFILEPARAMETER : L_MC1P_ProfileParameter;
END_VAR
END_METHOD

METHOD CALCPROFILE_80BC_CALCT5
VAR_INPUT
	LRSTARTACC : LREAL;
	LRSTARTVEL : LREAL;
	LRMAXACC : LREAL;
	LRMAXDEC : LREAL;
	LRMAXVEL : LREAL;
	LRTARGETACC : LREAL;
	LRTARGETVEL : LREAL;
	LRTARGETPOS : LREAL;
	LRMINPOSUNIT : LREAL;
	LRJERKACC : LREAL;
	LRJERKDEC : LREAL;
	LRJERKTIMEACC : LREAL;
	LRJERKTIMEDEC : LREAL;
	T01 : LREAL;
	T12 : LREAL;
	T23 : LREAL;
END_VAR
VAR_OUTPUT
	T5 : ARRAY [1..2] OF LREAL;
END_VAR
END_METHOD

METHOD CALCPROFILE_80BC_PROFILEDATA
VAR_INPUT
	LRSTARTACC : LREAL;
	LRSTARTVEL : LREAL;
	LRMAXACC : LREAL;
	LRMAXDEC : LREAL;
	LRMAXVEL : LREAL;
	LRTARGETACC : LREAL;
	LRTARGETVEL : LREAL;
	LRTARGETPOS : LREAL;
	LRJERKACC : LREAL;
	LRJERKDEC : LREAL;
	LRJERKTIMEACC : LREAL;
	LRJERKTIMEDEC : LREAL;
	T01 : LREAL;
	T12 : LREAL;
	T23 : LREAL;
	T5 : LREAL;
END_VAR
VAR_IN_OUT
	SCPROFILEDATA : L_MC1P_ProfileData;
END_VAR
END_METHOD

METHOD CALCPROFILE_80BD
VAR_INPUT
	LRSTARTACC : LREAL;
	LRSTARTVEL : LREAL;
	LRMAXACC : LREAL;
	LRMAXDEC : LREAL;
	LRMAXVEL : LREAL;
	LRTARGETACC : LREAL;
	LRTARGETVEL : LREAL;
	LRTARGETPOS : LREAL;
	LRJERKACC : LREAL;
	LRJERKDEC : LREAL;
	LRJERKTIMEACC : LREAL;
	LRJERKTIMEDEC : LREAL;
	SCMAXPROFILEDATA : L_MC1P_IntProfileData;
	SCMINPROFILEDATA : L_MC1P_IntProfileData;
END_VAR
VAR_OUTPUT
	DWSTATE : DWORD;
END_VAR
VAR_IN_OUT
	SCPROFILEDATA : L_MC1P_ProfileData;
	SCPROFILEPARAMETER : L_MC1P_ProfileParameter;
END_VAR
END_METHOD

METHOD CALCPROFILE_80BD_CALCT5
VAR_INPUT
	LRSTARTACC : LREAL;
	LRSTARTVEL : LREAL;
	LRMAXACC : LREAL;
	LRMAXDEC : LREAL;
	LRMAXVEL : LREAL;
	LRTARGETACC : LREAL;
	LRTARGETVEL : LREAL;
	LRTARGETPOS : LREAL;
	LRMINPOSUNIT : LREAL;
	LRJERKACC : LREAL;
	LRJERKDEC : LREAL;
	LRJERKTIMEACC : LREAL;
	LRJERKTIMEDEC : LREAL;
	T01 : LREAL;
	T12 : LREAL;
	T23 : LREAL;
END_VAR
VAR_OUTPUT
	T5 : ARRAY [1..2] OF LREAL;
END_VAR
END_METHOD

METHOD CALCPROFILE_80BD_PROFILEDATA
VAR_INPUT
	LRSTARTACC : LREAL;
	LRSTARTVEL : LREAL;
	LRMAXACC : LREAL;
	LRMAXDEC : LREAL;
	LRMAXVEL : LREAL;
	LRTARGETACC : LREAL;
	LRTARGETVEL : LREAL;
	LRTARGETPOS : LREAL;
	LRJERKACC : LREAL;
	LRJERKDEC : LREAL;
	LRJERKTIMEACC : LREAL;
	LRJERKTIMEDEC : LREAL;
	T01 : LREAL;
	T12 : LREAL;
	T23 : LREAL;
	T5 : LREAL;
END_VAR
VAR_IN_OUT
	SCPROFILEDATA : L_MC1P_ProfileData;
END_VAR
END_METHOD

METHOD CALCLINPROFILE_80C0
VAR_INPUT
	LRSTARTACC : LREAL;
	LRSTARTVEL : LREAL;
	SCPROFILEPARAMETER : L_MC1P_ProfileParameter;
	SCMINPROFILEDATA : L_MC1P_IntProfileData;
END_VAR
VAR_OUTPUT
	SCPROFILEDATA : L_MC1P_ProfileData;
END_VAR
END_METHOD

METHOD CALCPROFILE_80CA
VAR_INPUT
	LRSTARTACC : LREAL;
	LRSTARTVEL : LREAL;
	LRMAXACC : LREAL;
	LRMAXDEC : LREAL;
	LRMAXVEL : LREAL;
	LRTARGETACC : LREAL;
	LRTARGETVEL : LREAL;
	LRTARGETPOS : LREAL;
	LRJERKACC : LREAL;
	LRJERKDEC : LREAL;
	LRJERKTIMEACC : LREAL;
	LRJERKTIMEDEC : LREAL;
	SCMAXPROFILEDATA : L_MC1P_IntProfileData;
	SCMINPROFILEDATA : L_MC1P_IntProfileData;
END_VAR
VAR_OUTPUT
	DWSTATE : DWORD;
END_VAR
VAR_IN_OUT
	SCPROFILEDATA : L_MC1P_ProfileData;
	SCPROFILEPARAMETER : L_MC1P_ProfileParameter;
END_VAR
END_METHOD

METHOD CALCPROFILE_80CA_PROFILEDATA
VAR_INPUT
	LRSTARTACC : LREAL;
	LRSTARTVEL : LREAL;
	LRMAXACC : LREAL;
	LRMAXDEC : LREAL;
	LRMAXVEL : LREAL;
	LRTARGETACC : LREAL;
	LRTARGETVEL : LREAL;
	LRTARGETPOS : LREAL;
	LRJERKACC : LREAL;
	LRJERKDEC : LREAL;
	LRJERKTIMEACC : LREAL;
	LRJERKTIMEDEC : LREAL;
	T45 : LREAL;
	T56 : LREAL;
	T67 : LREAL;
END_VAR
VAR_IN_OUT
	SCPROFILEDATA : L_MC1P_ProfileData;
END_VAR
END_METHOD

METHOD CALCPROFILE_80CB
VAR_INPUT
	LRSTARTACC : LREAL;
	LRSTARTVEL : LREAL;
	LRMAXACC : LREAL;
	LRMAXDEC : LREAL;
	LRMAXVEL : LREAL;
	LRTARGETACC : LREAL;
	LRTARGETVEL : LREAL;
	LRTARGETPOS : LREAL;
	LRJERKACC : LREAL;
	LRJERKDEC : LREAL;
	LRJERKTIMEACC : LREAL;
	LRJERKTIMEDEC : LREAL;
	SCMAXPROFILEDATA : L_MC1P_IntProfileData;
	SCMINPROFILEDATA : L_MC1P_IntProfileData;
END_VAR
VAR_OUTPUT
	DWSTATE : DWORD;
END_VAR
VAR_IN_OUT
	SCPROFILEDATA : L_MC1P_ProfileData;
	SCPROFILEPARAMETER : L_MC1P_ProfileParameter;
END_VAR
END_METHOD

METHOD CALCPROFILE_80CB_PROFILEDATA
VAR_INPUT
	LRSTARTACC : LREAL;
	LRSTARTVEL : LREAL;
	LRMAXACC : LREAL;
	LRMAXDEC : LREAL;
	LRMAXVEL : LREAL;
	LRTARGETACC : LREAL;
	LRTARGETVEL : LREAL;
	LRTARGETPOS : LREAL;
	LRJERKACC : LREAL;
	LRJERKDEC : LREAL;
	LRJERKTIMEACC : LREAL;
	LRJERKTIMEDEC : LREAL;
	T45 : LREAL;
	T56 : LREAL;
	T67 : LREAL;
END_VAR
VAR_IN_OUT
	SCPROFILEDATA : L_MC1P_ProfileData;
END_VAR
END_METHOD

METHOD CALCPROFILE_80CC
VAR_INPUT
	LRSTARTACC : LREAL;
	LRSTARTVEL : LREAL;
	LRMAXACC : LREAL;
	LRMAXDEC : LREAL;
	LRMAXVEL : LREAL;
	LRTARGETACC : LREAL;
	LRTARGETVEL : LREAL;
	LRTARGETPOS : LREAL;
	LRJERKACC : LREAL;
	LRJERKDEC : LREAL;
	LRJERKTIMEACC : LREAL;
	LRJERKTIMEDEC : LREAL;
	SCMAXPROFILEDATA : L_MC1P_IntProfileData;
	SCMINPROFILEDATA : L_MC1P_IntProfileData;
END_VAR
VAR_OUTPUT
	DWSTATE : DWORD;
END_VAR
VAR_IN_OUT
	SCPROFILEDATA : L_MC1P_ProfileData;
	SCPROFILEPARAMETER : L_MC1P_ProfileParameter;
END_VAR
END_METHOD

METHOD CALCPROFILE_80CC_PROFILEDATA
VAR_INPUT
	LRSTARTACC : LREAL;
	LRSTARTVEL : LREAL;
	LRMAXACC : LREAL;
	LRMAXDEC : LREAL;
	LRMAXVEL : LREAL;
	LRTARGETACC : LREAL;
	LRTARGETVEL : LREAL;
	LRTARGETPOS : LREAL;
	LRJERKACC : LREAL;
	LRJERKDEC : LREAL;
	LRJERKTIMEACC : LREAL;
	LRJERKTIMEDEC : LREAL;
	T45 : LREAL;
	T56 : LREAL;
	T67 : LREAL;
END_VAR
VAR_IN_OUT
	SCPROFILEDATA : L_MC1P_ProfileData;
END_VAR
END_METHOD

METHOD CALCPROFILE_80CD
VAR_INPUT
	LRSTARTACC : LREAL;
	LRSTARTVEL : LREAL;
	LRMAXACC : LREAL;
	LRMAXDEC : LREAL;
	LRMAXVEL : LREAL;
	LRTARGETACC : LREAL;
	LRTARGETVEL : LREAL;
	LRTARGETPOS : LREAL;
	LRJERKACC : LREAL;
	LRJERKDEC : LREAL;
	LRJERKTIMEACC : LREAL;
	LRJERKTIMEDEC : LREAL;
	SCMAXPROFILEDATA : L_MC1P_IntProfileData;
	SCMINPROFILEDATA : L_MC1P_IntProfileData;
END_VAR
VAR_OUTPUT
	DWSTATE : DWORD;
END_VAR
VAR_IN_OUT
	SCPROFILEDATA : L_MC1P_ProfileData;
	SCPROFILEPARAMETER : L_MC1P_ProfileParameter;
END_VAR
END_METHOD

METHOD CALCPROFILE_80CD_CALCT3
VAR_INPUT
	LRSTARTACC : LREAL;
	LRSTARTVEL : LREAL;
	LRMAXACC : LREAL;
	LRMAXDEC : LREAL;
	LRMAXVEL : LREAL;
	LRTARGETACC : LREAL;
	LRTARGETVEL : LREAL;
	LRTARGETPOS : LREAL;
	LRMINPOSUNIT : LREAL;
	LRJERKACC : LREAL;
	LRJERKDEC : LREAL;
	LRJERKTIMEACC : LREAL;
	LRJERKTIMEDEC : LREAL;
	T45 : LREAL;
	T56 : LREAL;
	T67 : LREAL;
END_VAR
VAR_OUTPUT
	T3 : ARRAY [1..2] OF LREAL;
END_VAR
END_METHOD

METHOD CALCPROFILE_80CD_PROFILEDATA
VAR_INPUT
	LRSTARTACC : LREAL;
	LRSTARTVEL : LREAL;
	LRMAXACC : LREAL;
	LRMAXDEC : LREAL;
	LRMAXVEL : LREAL;
	LRTARGETACC : LREAL;
	LRTARGETVEL : LREAL;
	LRTARGETPOS : LREAL;
	LRJERKACC : LREAL;
	LRJERKDEC : LREAL;
	LRJERKTIMEACC : LREAL;
	LRJERKTIMEDEC : LREAL;
	T45 : LREAL;
	T56 : LREAL;
	T67 : LREAL;
	T3 : LREAL;
END_VAR
VAR_IN_OUT
	SCPROFILEDATA : L_MC1P_ProfileData;
END_VAR
END_METHOD

(* ---- L_MC1P_POSPROFILERCLUTCH.pou ---- *)
FUNCTION_BLOCK L_MC1P_POSPROFILERCLUTCH
VAR_INPUT
	XENABLE : BOOL;
	XSYNCPOS : BOOL;
	XEXECUTEGAP : BOOL;
	XAUXEXECUTEGAP : BOOL;
	LRTASKCYCLETIME : LREAL := 0.001;
	LRSLAVESYNCOUTPOS : LREAL;
	LRCYCMASTERPOS : LREAL;
	LRCYCMASTERVEL : LREAL;
	LRCYCMASTERACC : LREAL;
	LRSETSLAVEPOS : LREAL;
	LRSETSLAVEVEL : LREAL;
	LRSETSLAVEACC : LREAL;
	LRJERK : LREAL := 10000;
	LRMAXACC : LREAL := 100;
	LRMAXDEC : LREAL := 100;
	LRMAXVEL : LREAL := 10;
	FB_POSPROFILERPOS : REFERENCE TO L_MC1P_PosProfiler;
END_VAR
VAR_OUTPUT
	XBUSY : BOOL;
	XDONE : BOOL;
	XACCDECSYNC : BOOL;
	XPOSSYNCHRONISED : BOOL;
	XERROR : BOOL;
	EERRORID : WORD;
	LRSETSLAVEPOSOUT : LREAL;
	LRSETSLAVEVELOUT : LREAL;
	LRSETSLAVEACCOUT : LREAL;
END_VAR
VAR
	SCPROFILEPARAMETER : L_MC1P_ProfileParameter;
	WSTEPPER : WORD;
	XEXECUTEPOSPROFILER : BOOL;
	LRSLAVESYNCOUTPOS_INT : LREAL;
	XAUXEXECUTEPROFILE : BOOL;
	XEXECUTEPROFILE : BOOL;
	LRSETPOSPROFILER : LREAL;
	LRSETACCPROFILER : LREAL;
	LRSETVELPROFILER : LREAL;
	LRCYCMASTERPOS_INT : LREAL;
	LRCYCMASTERVEL_INT : LREAL;
	LRCYCMASTERACC_INT : LREAL;
	XPOSSYNCHRONISED_INT : BOOL;
	XEXECUTEGAPOLD : BOOL;
	XAUXEXECUTEGAPOLD : BOOL;
	XENABLEOLD : BOOL;
	LRCYCMASTERPOS_OLD : LREAL;
	LRTOLERANCE : LREAL;
END_VAR
END_FUNCTION_BLOCK

METHOD CALL_ERRORHANDLER
END_METHOD

METHOD CALL_FBMETHODES
END_METHOD

METHOD CALL_FB_POSPROFILERPOS
END_METHOD

METHOD CALL_FB_POSPROFILERPOSINPUTS
END_METHOD

METHOD CALL_OUTPUTS
END_METHOD

METHOD CALL_PROFILEPARAMETER
END_METHOD

METHOD CALL_RESETCOMMANDS
END_METHOD

METHOD CALL_RESETOUTPUTS
END_METHOD

METHOD CALL_STATEMACHINE
END_METHOD

(* ---- L_MC1P_POSPROFILERCLUTCHSTATE.pou ---- *)
FUNCTION_BLOCK L_MC1P_POSPROFILERCLUTCHSTATE EXTENDS L_MC1P_PosProfilerClutch
VAR_INPUT
	XSYNCOUTINSTANT : BOOL;
	XMOVETOTARGETPOS : BOOL;
	LRTARGETPOS : LREAL;
	EDIRECTION : INT := 0;
	LRAXESCYCLELENGTH : LREAL := 360;
	EAXESTRAVERSINGRANGE : L_MC1P_TraversingRange;
	LRPOSITIONINGJERK : LREAL;
	LRPOSITIONINGACC : LREAL;
	LRPOSITIONINGDEC : LREAL;
	LRPOSITIONINGVEL : LREAL;
	LRSYNCOUTINSTANTJERK : LREAL;
	LRSYNCOUTINSTANTDEC : LREAL;
END_VAR
VAR_OUTPUT
	XREVERSING : BOOL;
	XPOSITIONING : BOOL;
	XINPOSITION : BOOL;
END_VAR
VAR
	XREVERSING_INT : BOOL;
	WMODE : WORD;
	XSYNCOUTINSTANT_OLD : BOOL;
	XMOVETOTARGETPOS_OLD : BOOL;
	XPOSMODE_INT : BOOL;
	LRTASKCYCLETIME_INT : LREAL;
	LRAXESCYCLELENGTH_INT : LREAL;
	LRTARGETPOS_INT : LREAL;
	LRTARGETPOS_LOCK : LREAL;
	LRTOLERANCEVEL : LREAL;
	LRTOLERANCEACC : LREAL;
	LRACCDIST : LREAL;
	XVELTRACE : BOOL;
	WVELTRACESTEPPER : WORD;
	LRSETACC_PROFILERPOS : LREAL;
	LRPOSPROFILERSPEED_ABS : LREAL;
	WREVERSINGVELMODE : WORD;
	LRVELZERROTOLERANZ : LREAL;
	LRSETSLAVEVELOUT_OLD : LREAL;
END_VAR
END_FUNCTION_BLOCK

METHOD CALL_CALCTARGETPOS
VAR_INPUT
	LRTARGETPOS : LREAL;
END_VAR
END_METHOD

METHOD CALL_CALCTOLERANCE
END_METHOD

METHOD CALL_CALCLRCYCMASTERPOS
END_METHOD

METHOD CALL_ERRORHANDLER
END_METHOD

METHOD CALL_FBMETHODES
END_METHOD

METHOD CALL_FB_POSPROFILERPOS
END_METHOD

METHOD CALL_FB_POSPROFILERPOSINPUTS
END_METHOD

METHOD CALL_OUTPUTS
END_METHOD

METHOD CALL_PROFILEPARAMETER
END_METHOD

METHOD CALL_PROFILEPARAMETERACCDECINMODE2
END_METHOD

METHOD CALL_RESETCOMMANDS
END_METHOD

METHOD CALL_RESETOUTPUTS
END_METHOD

METHOD CALL_STATEMACHINE
END_METHOD

(* ---- L_MC1P_POSPROFILEROPTDECUSAGE.pou ---- *)
FUNCTION_BLOCK L_MC1P_POSPROFILEROPTDECUSAGE
VAR
	PPOSPROFILER : POINTER TO L_MC1P_PosProfiler;
	SCPROFILEDATAEXTENDED : L_MC1P_ProfileDataExtended;
	LRTASKCYCLE : LREAL;
	LRINVTASKCYCLE : LREAL;
	XEXTENDEDPROFILEVALID : BOOL;
	WCALCPROFILEMODE : REFERENCE TO WORD;
	WCALCPROFILESTEP : REFERENCE TO WORD;
	PROFILEPHASE : REFERENCE TO L_MC1P_ProfilePhaseData;
	XCALCPROFILEACTIVE : REFERENCE TO BOOL;
	XPROFILECALCULATED : REFERENCE TO BOOL;
	XCALCPROFILEDATAACTIVE : REFERENCE TO BOOL;
	XSEARCHTIMES1_DONE : REFERENCE TO BOOL;
	XSEARCHTIMESACTIVE : REFERENCE TO BOOL;
	SIGNOFMAXVEL : REFERENCE TO LREAL;
	WITERATIONCYCLESLIMIT1 : REFERENCE TO WORD;
	S_MIN : REFERENCE TO LREAL;
	INITPHASEDATA : REFERENCE TO L_MC1P_ProfilePhaseData;
	DWMINPROFILETYPE : REFERENCE TO DWORD;
	XUSESTARTJERK : REFERENCE TO BOOL;
	LRMINREFJERK : REFERENCE TO LREAL;
	LRACTPROFILEJERK : REFERENCE TO LREAL;
	PROVISIONALPROFILE : REFERENCE TO L_MC1P_IntProfileData;
	PROVISIONALPROFILEOLD : REFERENCE TO L_MC1P_IntProfileData;
	S_PROVISIONALPROFILE : REFERENCE TO LREAL;
	LRACTPROFILETIME : REFERENCE TO LREAL;
	XERROR : REFERENCE TO BOOL;
	JERKACCTEMP1 : REFERENCE TO LREAL;
	JERKACCTEMP2 : REFERENCE TO LREAL;
	VELPHASE4 : REFERENCE TO LREAL;
	MINVELPHASE4 : REFERENCE TO LREAL;
	XPHASE0FINISHED : REFERENCE TO BOOL;
	VMAXMINTRIACC1 : REFERENCE TO LREAL;
	VMAXMINTRIACC2 : REFERENCE TO LREAL;
	MAXPROFILEPHASEINDEX : WORD := 10;
END_VAR
END_FUNCTION_BLOCK

METHOD CALCPROFILEDATA
VAR_INPUT
	PPOSPROFILERDATA : POINTER TO L_MC1P_PosProfiler;
	LRSTARTACC : LREAL;
	LRSTARTVEL : LREAL;
	LRSTARTPOS : LREAL;
	XVELMODE : BOOL;
END_VAR
VAR_OUTPUT
	XERROR : BOOL;
	DWSTATE : DWORD;
	DWPROFILETYPE : DWORD;
END_VAR
VAR_IN_OUT
	SCPROFILEDATA : L_MC1P_ProfileData;
	SCPROFILEPARAMETER : L_MC1P_ProfileParameter;
END_VAR
END_METHOD

METHOD CALCPROVISIONALPROFILEDATAOPTDECUSAGE : BOOL
VAR_IN_OUT
	LRSTARTPOS : LREAL;
	LRSTARTVEL : LREAL;
	LRSTARTACC : LREAL;
	LRSTARTVELINT : LREAL;
	LRSTARTACCINT : LREAL;
	LRRECIPRJERKACC : LREAL;
	LRRECIPRJERKDEC : LREAL;
	SCPROFILEPARAMETERINT : L_MC1P_ProfileParameter;
	XVELMODE : BOOL;
	SIGNOFMAXVEL : LREAL;
	DWPROFILETYPE : DWORD;
	DWMINPOSPROFILETYPE : DWORD;
	XCALCPROFILE : BOOL;
	WCALCPROFILESTEP : WORD;
	XPOSITIVEMOVEMENT : BOOL;
	SCPROFILEDATAPHASE0 : L_MC1P_ProfilePhaseData;
	SCPROFILEDATAREVPHASE : L_MC1P_IntProfileDataAcc;
	SCPROFILEDATA : L_MC1P_ProfileData;
	DWSTATECALCPROFILE : DWORD;
	SCMAXPROFILEDATA : L_MC1P_IntProfileData;
	SCMINPROFILEDATA : L_MC1P_IntProfileData;
END_VAR
END_METHOD

METHOD CHECKPROFILEDATA
VAR_INPUT
	DWMODE : DWORD;
	LRTARGETPOS : LREAL;
	LRTARGETVEL : LREAL;
	LRTARGETACC : LREAL;
	LRJERKPHASE7 : LREAL;
END_VAR
VAR_OUTPUT
	XERROR : BOOL;
END_VAR
VAR_IN_OUT
	SCPROFILEDATA : L_MC1P_ProfileDataExtended;
END_VAR
END_METHOD

METHOD PROFILEINTERPOLATOR : BOOL
VAR_INPUT
	PPOSPROFILERDATA : POINTER TO L_MC1P_PosProfiler;
	LREVALTIME : LREAL;
END_VAR
VAR_OUTPUT
	DWSTATE : DWORD;
	LRSETPOS : LREAL;
	LRSETVEL : LREAL;
	LRSETACC : LREAL;
END_VAR
VAR_IN_OUT
	SCPROFILEDATA : L_MC1P_ProfileData;
END_VAR
END_METHOD

METHOD SETPROFILERINSTANCE : BOOL
END_METHOD

METHOD STRETCHPROFILE
VAR_INPUT
	PPOSPROFILERDATA : POINTER TO L_MC1P_PosProfiler;
	LRTIMEBASE : LREAL;
END_VAR
VAR_IN_OUT
	SCPROFILEDATA : L_MC1P_ProfileData;
END_VAR
END_METHOD

(* ---- L_MC1P_POSRECONSTRUCTION.pou ---- *)
FUNCTION_BLOCK L_MC1P_POSRECONSTRUCTION
VAR_INPUT
	ETHCSLAVE : POINTER TO ETCSlave;
	XISABSOLUTEENCODER : BOOL := FALSE;
	XEXECUTEPOSITIONRESET : BOOL := FALSE;
	LRMAXPOSITIONDIFF : LREAL := 360;
	XIGNOREMTOFFSET : BOOL;
END_VAR
VAR_IN_OUT
	ENCODER : _AXIS_REF_ENC;
END_VAR
VAR
	RETAINDATA : L_MC1P_retainDataEncAxis;
	PXDUMMY : POINTER TO BOOL := 0;
	PRETAINDATA : POINTER TO L_MC1P_uRetainData;
	XHOMEPOSAVAILABLE : BOOL := FALSE;
	XMIRROR : BOOL := FALSE;
	WINITSTEP : WORD := 0;
	XENCODERPOSVALID : BOOL := FALSE;
	XENCODERPOSVALIDOLD : BOOL := FALSE;
	XETCSLAVEACTIVE : BOOL := FALSE;
	XEXECUTEPOSITIONRESETOLD : BOOL := FALSE;
	PLRDUMMY : POINTER TO LREAL;
	XETHCISACTIVE : BOOL;
	WETCSTATEOLD : WORD;
	AWCSTATE : ARRAY [0..3] OF BOOL;
	WSTATEWCCNT : WORD := 0;
	XBUSSECTIONINACTIVE : BOOL := FALSE;
	XINVALIDPOSITION : BOOL := FALSE;
	LRACTPOSOLD : LREAL := 0;
	DIENCODERPOSITIONOLD : DINT := 0;
	DITEST : DINT := 0;
	DITEST2 : DINT := 0;
	XIGNOREMTOFFSETINT : BOOL := FALSE;
	PRETAINHANDLING : POINTER TO L_MC1P_IRetainHandling;
	RETAINHANDLINGEXTFB : L_MC1P_MotionUtilsRetainHandlingExtFb;
	PWDUMMY : POINTER TO WORD;
	PIDUMMY : POINTER TO INT;
	IGNOREMTOFFSET : BOOL;
END_VAR
END_FUNCTION_BLOCK

(* ---- L_MC1P_POSSIGNALPROCESSING.pou ---- *)
FUNCTION_BLOCK L_MC1P_POSSIGNALPROCESSING
VAR_INPUT
	XENABLE : BOOL;
	DWSAMPERATE : DWORD;
END_VAR
VAR_OUTPUT
	DIPOSOUT : DINT;
	DIVELOUT : DINT;
	DIVELOUTDIFF : DINT;
	DIPOSIN : DINT;
	DWSAMPLETIME : DWORD;
	DWACTTIME : DWORD;
END_VAR
VAR
	LRCALLTIME : LREAL;
	LRTASKCYCLE : LREAL;
	XNEWVALUE : BOOL;
	DIACTPOSOLD : DINT;
	DWLASTTIMESTAMP : DWORD;
	DIPOSOUTOLD : DINT;
	XENABLEOLD : BOOL;
	XFIRSTCHANGELONGTIME : BOOL;
	DWTIMEDIFF : DWORD;
	DISPEEDRES : DINT;
	XDUMMY : BOOL;
END_VAR
END_FUNCTION_BLOCK

METHOD CALCVEL : DINT
VAR_INPUT
	POSDIFF : DINT;
	TIMEDIFF : DWORD;
END_VAR
VAR_IN_OUT
	AXIS : _AXIS_REF_REAL;
END_VAR
END_METHOD

METHOD CALCULATE : DINT
VAR_INPUT
	DIACTPOS : DINT;
	DWSAMPLETIME : DWORD;
	DWACTTIME : DWORD;
END_VAR
VAR_OUTPUT
	DIPOSOUT : DINT;
	XVELVALID : BOOL;
	DIVELOUT : DINT;
END_VAR
VAR_IN_OUT
	AXIS : _AXIS_REF_REAL;
END_VAR
END_METHOD

METHOD CHECKUPDATETIME : BOOL
END_METHOD

METHOD RESET
END_METHOD

(* ---- L_MC1P_POWER_INTERNAL.pou ---- *)
FUNCTION_BLOCK L_MC1P_POWER_INTERNAL EXTENDS L_MC1P_Template_Internal
VAR_OUTPUT
	STATUS : BOOL;
	VALID : BOOL;
	ERROR : BOOL;
	ERRORID : L_IE1P_Error;
	WACTIVEID : WORD := 0;
END_VAR
VAR
	XSWITCHONLOCKED : BOOL := FALSE;
	XDRIVEENABLELDOLD : BOOL := FALSE;
	XENABLEOLD : BOOL := FALSE;
	XENABLEREQUESTOLD : BOOL := FALSE;
	OBSERVE : TON;
	EOLDSTATE : L_MC1P_AXIS_STATE;
	XPLNOTVALID : BOOL := FALSE;
END_VAR
END_FUNCTION_BLOCK

METHOD MAIN
VAR_INPUT
	ENABLE : BOOL;
	ENABLEPOSITIVE : BOOL := TRUE;
	ENABLENEGATIVE : BOOL := TRUE;
END_VAR
VAR_OUTPUT
	XEXTERROR : BOOL;
	XEXTERRORID : L_IE1P_Error;
	XEXTSTATUS : BOOL;
	XEXTVALID : BOOL;
END_VAR
VAR_IN_OUT
	AXIS : AXIS_REF;
	WFBID : WORD;
END_VAR
END_METHOD

METHOD RESETACTIVEINSTANCE : WORD
END_METHOD

METHOD SETACTIVEINSTANCE : WORD
END_METHOD

(* ---- L_MC1P_PROFILEGENERATOR.pou ---- *)
FUNCTION_BLOCK L_MC1P_PROFILEGENERATOR
VAR_INPUT
	SCPROFILEPARAMETER : L_MC1P_ProfileParameter;
	XEXECUTE : BOOL := FALSE;
	XAUXEXECUTE : BOOL := FALSE;
	XABORT : BOOL := FALSE;
	XVELMODE : BOOL := FALSE;
	LRSTARTPOS : LREAL := 0.0;
	LRSTARTVEL : LREAL := 0.0;
	LRSTARTACC : LREAL := 0.0;
END_VAR
VAR_OUTPUT
	XDONE : BOOL;
	XBUSY : BOOL;
	XABORTED : BOOL;
	XERROR : BOOL;
	EERRORID : L_IE1P_Error;
	LRSETPOSOUT : LREAL;
	LRSETVELOUT : LREAL;
	LRSETACCOUT : LREAL;
END_VAR
VAR
	L_MC1P_POSPROFILER1 : L_MC1P_PosProfiler := STRUCT(wCalcProfileMode := 1);
	LRTASKCYCLE : LREAL := 0;
	LRINVTASKCYCLE : LREAL := 0;
	XERROROLD : BOOL;
	ALRDUMMY : ARRAY [0..8] OF LREAL := [9(0)];
	PROFILEPHASESTIME : ARRAY [0..8] OF LREAL;
	PROFILETIME : TIME;
	REMAININGTIMEOFPROFILE : LREAL;
	REMAININGTIMEOFPROFILEAVAILABLE : BOOL;
END_VAR
END_FUNCTION_BLOCK

(* ---- L_MC1P_RAMPGENERATOR.pou ---- *)
FUNCTION_BLOCK L_MC1P_RAMPGENERATOR
VAR_INPUT
	LRSETVEL : LREAL;
	LRACC : LREAL;
	LRDEC : LREAL;
	LRJERK : LREAL;
	XLOADSTARTVALUE : BOOL;
	LRSTARTVALUE : LREAL;
END_VAR
VAR_OUTPUT
	LRSETVELOUT : LREAL;
	LRSETACCDECOUT : LREAL;
END_VAR
VAR
	FBRAMPGENERATOR : L_MC1P_HlpRampGenerator;
END_VAR
END_FUNCTION_BLOCK

(* ---- L_MC1P_RAMPGENERATORINTERN.pou ---- *)
FUNCTION_BLOCK L_MC1P_RAMPGENERATORINTERN
VAR_INPUT
	LRACC : LREAL := 0;
	LRDEC : LREAL := 0;
	LRVEL : LREAL := 0;
	LRJERKACC : LREAL := 0;
	LRJERKDEC : LREAL := 0;
	LRTASKCYCLE : LREAL := 0;
	XRESET : BOOL := FALSE;
END_VAR
VAR_OUTPUT
	LRSETPOS : LREAL := 0;
	LRSETVEL : LREAL := 0;
	LRSETACCDEC : LREAL := 0;
	DNSTATE : DINT := 0;
	C_RG_STATE_INI : DINT := 0;
	C_RG_STATE_CNS : DINT := 1;
	C_RG_STATE_ACC : DINT := 2;
	C_RG_STATE_DEC : DINT := 3;
END_VAR
VAR
	XINITIALIZED : BOOL := FALSE;
	FBHLPRAMPGENERATOR : L_MC1P_HlpRampGenerator;
END_VAR
END_FUNCTION_BLOCK

METHOD SETSTARTVALUES
VAR_INPUT
	LRVEL : LREAL := 0;
	LRACC : LREAL := 0;
	LRTASKCYCLE : LREAL := 0;
END_VAR
END_METHOD

(* ---- L_MC1P_READAXISERROR_INTERNAL.pou ---- *)
FUNCTION_BLOCK L_MC1P_READAXISERROR_INTERNAL EXTENDS L_MC1P_Template_IntFB
VAR_INPUT
	ENABLE : BOOL;
END_VAR
VAR_OUTPUT
	VALID : BOOL;
	BUSY : BOOL;
	ERROR : BOOL;
	ERRORID : L_IE1P_Error;
	AXISWARNING : BOOL;
	AXISERROR : BOOL;
	AXISERRORID : L_IE1P_Error;
	PINSTANCENAME : POINTER TO STRING;
	TIMESTAMP : TIME;
	DRIVEWARNING : BOOL;
	DRIVEERROR : BOOL;
	DRIVEERRORID : DWORD;
END_VAR
VAR
	XENABLEOLD : BOOL;
	READPARAMETER : L_MC1P_ReadParameter_Internal;
	PAXIS : POINTER TO _AXIS_REF_REAL;
	NOERROR : STRING := '';
	UNDEFERROR : STRING := 'undefined';
END_VAR
END_FUNCTION_BLOCK

METHOD MAIN
VAR_IN_OUT
	AXIS : AXIS_REF;
	FBBASE : L_MC1P_Template_ForAxis;
END_VAR
END_METHOD

(* ---- L_MC1P_READAXISINFO_INTERNAL.pou ---- *)
FUNCTION_BLOCK L_MC1P_READAXISINFO_INTERNAL EXTENDS L_MC1P_Template_IntFB
VAR_INPUT
	ENABLE : BOOL;
END_VAR
VAR_OUTPUT
	VALID : BOOL;
	BUSY : BOOL;
	ERROR : BOOL;
	ERRORID : L_IE1P_Error;
	HOMEABSSWITCH : BOOL;
	LIMITSWITCHPOS : BOOL;
	LIMITSWITCHNEG : BOOL;
	SIMULATION : BOOL;
	COMMUNICATIONREADY : BOOL;
	READYFORPOWERON : BOOL;
	POWERON : BOOL;
	ISHOMED : BOOL;
	AXISERROR : BOOL;
	AXISWARNING : BOOL;
	DRIVEWARNING : BOOL;
	DRIVEERROR : BOOL;
	SWLIMITSWITCHPOS : BOOL;
	SWLIMITSWITCHNEG : BOOL;
	READYFORMOTION : BOOL;
	STOACTIVE : BOOL;
	VOLTAGEENABLED : BOOL;
	MOTORMAGNETISED : BOOL;
	QSPAPPLACTIVE : BOOL;
	QSPDRIVEACTIVE : BOOL;
END_VAR
VAR
	XENABLEOLD : BOOL;
END_VAR
END_FUNCTION_BLOCK

METHOD MAIN
VAR_IN_OUT
	AXIS : AXIS_REF;
	FBBASE : L_MC1P_Template_ForAxis;
END_VAR
END_METHOD

(* ---- L_MC1P_READAXISSTATUSWORDS.pou ---- *)
FUNCTION_BLOCK L_MC1P_READAXISSTATUSWORDS EXTENDS L_MC1P_Template
VAR_INPUT
	XENABLE : BOOL;
END_VAR
VAR_OUTPUT
	XVALID : BOOL;
	XBUSY : BOOL;
	XERROR : BOOL;
	EERRORID : L_IE1P_Error;
	WCIA402STATUSWORD : WORD;
	WLENZESTATUSWORD : WORD;
	WLENZESTATUSWORD2 : WORD;
END_VAR
VAR
	XENABLEOLD : BOOL;
END_VAR
END_FUNCTION_BLOCK

(* ---- L_MC1P_READMACHINEDATA.pou ---- *)
FUNCTION_BLOCK L_MC1P_READMACHINEDATA EXTENDS L_MC1P_Template
VAR_INPUT
	XENABLE : BOOL;
END_VAR
VAR_OUTPUT
	XVALID : BOOL;
	XBUSY : BOOL;
	XERROR : BOOL;
	EERRORID : L_IE1P_Error;
	LRFEEDCONSTANT : LREAL;
	DWGEARDENOMINATOR : DWORD;
	DWGEARNUMERATOR : DWORD;
	DWADDGEARDENOMINATOR : DWORD;
	DWADDGEARNUMERATOR : DWORD;
	DWPOSRESOLUTION : DWORD;
	XORIENTATION : BOOL;
	ETRAVERSINGRANGE : L_MC1P_TraversingRange;
	LRCYCLELENGTH : LREAL;
	XVIRTUAL : BOOL;
END_VAR
VAR
	XENABLEOLD : BOOL;
	PAXIS : POINTER TO _AXIS_REF_REAL;
END_VAR
END_FUNCTION_BLOCK

(* ---- L_MC1P_READMOTIONSTATE_INTERNAL.pou ---- *)
FUNCTION_BLOCK L_MC1P_READMOTIONSTATE_INTERNAL EXTENDS L_MC1P_Template_IntFB
VAR_INPUT
	ENABLE : BOOL;
	SOURCE : MC_SOURCE;
END_VAR
VAR_OUTPUT
	VALID : BOOL;
	BUSY : BOOL;
	ERROR : BOOL;
	ERRORID : L_IE1P_Error;
	CONSTANTVELOCITY : BOOL;
	ACCELERATING : BOOL;
	DECELERATING : BOOL;
	DIRECTIONPOSITIVE : BOOL;
	DIRECTIONNEGATIVE : BOOL;
	INPOSITION : BOOL;
	STANDSTILLSETVELOCITY : BOOL;
	STANDSTILLACTVELOCITY : BOOL;
END_VAR
VAR
	XENABLEOLD : BOOL;
	LRACTVELOCITYOLD : LREAL;
	LRSETVELOCITYOLD : LREAL;
	XDRIVEENABLEDOLD : BOOL;
	LRTEMP : LREAL;
	LRTEMPABS : LREAL;
	SOURCEINT : MC_SOURCE;
END_VAR
END_FUNCTION_BLOCK

METHOD MAIN
VAR_IN_OUT
	AXIS : AXIS_REF;
	FBBASE : L_MC1P_Template_ForAxis;
END_VAR
END_METHOD

(* ---- L_MC1P_READPARAMETER_INTERNAL.pou ---- *)
FUNCTION_BLOCK L_MC1P_READPARAMETER_INTERNAL EXTENDS L_MC1P_Template_IntFB
VAR_INPUT
	ENABLE : BOOL;
	PARAMETERNUMBER : DINT;
	TCYCLETIME : TIME := TIME#1ms;
END_VAR
VAR_OUTPUT
	VALID : BOOL;
	BUSY : BOOL;
	ERROR : BOOL;
	ERRORID : L_IE1P_Error;
	VALUE : LREAL;
END_VAR
VAR
	XENABLEOLD : BOOL := FALSE;
	PARAMETERNUMBEROLD : DINT := 0;
	L_DCO_READDRIVEPARAMETER1 : L_DCO_ReadDriveParameter;
	TIMERREADCYCLE : TON;
	DATA : L_DCO_ConvertData;
	XERRORHOLD : BOOL;
	EERRORIDHOLD : L_IE1P_Error;
	DWPARAMETERNUMBERINT : DWORD;
END_VAR
END_FUNCTION_BLOCK

METHOD MAIN
VAR_IN_OUT
	AXIS : AXIS_REF;
	FBBASE : L_MC1P_Template_ForAxis;
END_VAR
END_METHOD

METHOD FB_RESET : BOOL
END_METHOD

(* ---- L_MC1P_READSETPOSITION.pou ---- *)
FUNCTION_BLOCK L_MC1P_READSETPOSITION EXTENDS L_MC1P_Template
VAR_INPUT
	XENABLE : BOOL;
END_VAR
VAR_OUTPUT
	XVALID : BOOL;
	XBUSY : BOOL;
	XERROR : BOOL;
	EERRORID : L_IE1P_Error;
	LRPOSITION : LREAL;
END_VAR
VAR
	XENABLEOLD : BOOL;
END_VAR
END_FUNCTION_BLOCK

(* ---- L_MC1P_REINITALLNODES.pou ---- *)
FUNCTION_BLOCK L_MC1P_REINITALLNODES
VAR_INPUT
	XEXECUTE : BOOL;
	XINITCOMMUNICATION : BOOL := TRUE;
END_VAR
VAR_OUTPUT
	XDONE : BOOL;
	XBUSY : BOOL;
	XERROR : BOOL;
	EERRORID : L_IE1P_Error;
END_VAR
VAR
	PAXIS : POINTER TO AXIS_REF;
	DIIDX : DINT;
	ISTEP : INT;
	PWDUMMY : POINTER TO WORD;
	XERROR_INT : BOOL;
	XDONE_INT : BOOL;
	XRESETOUTPUT : BOOL;
	XEXECUTEOLD : BOOL;
	XREALAXISAVAILABLE : BOOL;
	DIFIRSTREALAXISINIT : DINT;
	_EERRORID : L_IE1P_Error := L_IE1P_Error.NoError;
	XNOCOMMAXISDETECTED : BOOL;
	PSLAVE : POINTER TO ETCSlave;
	PMASTER : POINTER TO L_IODrvEtherCAT;
	WMASTERSTATE : WORD;
END_VAR
END_FUNCTION_BLOCK

(* ---- L_MC1P_REINITNODE.pou ---- *)
FUNCTION_BLOCK L_MC1P_REINITNODE EXTENDS L_MC1P_Template
VAR_INPUT
	XEXECUTE : BOOL;
END_VAR
VAR_OUTPUT
	XDONE : BOOL;
	XBUSY : BOOL;
	XERROR : BOOL;
	EERRORID : L_IE1P_Error;
END_VAR
VAR
	XEXECUTEOLD : BOOL;
	XRESETOUTPUT : BOOL;
	PWDUMMY : POINTER TO WORD;
	RESET : MC_Reset;
	XRESET : BOOL;
END_VAR
END_FUNCTION_BLOCK

(* ---- L_MC1P_RESET_INTERNAL.pou ---- *)
FUNCTION_BLOCK L_MC1P_RESET_INTERNAL EXTENDS L_MC1P_Template_IntFB
VAR_INPUT
	EXECUTE : BOOL;
END_VAR
VAR_OUTPUT
	DONE : BOOL;
	BUSY : BOOL;
	ERROR : BOOL;
	ERRORID : L_IE1P_Error;
END_VAR
VAR
	XEXECUTEOLD : BOOL;
	PITMP : POINTER TO INT;
	XRESETOUTPUT : BOOL;
	PXDUMMY : POINTER TO BOOL;
	DWRESETCYCLEDRIVEERROR : DWORD;
	DWRESETCYCLECOUNTERSTART : DWORD;
	DWMAXTIMEOUT : DWORD;
	XRESETPOSSIBLE : BOOL;
	PERRORINFO : POINTER TO L_MC1P_ErrorInformation;
	XWAITFORRESETEVENT : BOOL;
	XSENDREQUESTRESET : BOOL;
	XRESETDRIVE : BOOL;
END_VAR
END_FUNCTION_BLOCK

METHOD MAIN
VAR_IN_OUT
	AXIS : AXIS_REF;
	FBBASE : L_MC1P_Template_ForAxis;
END_VAR
END_METHOD

(* ---- L_MC1P_RESETFOLLOWINGERROR.pou ---- *)
FUNCTION_BLOCK L_MC1P_RESETFOLLOWINGERROR EXTENDS L_MC1P_Template
VAR_INPUT
	XEXECUTE : BOOL;
END_VAR
VAR_OUTPUT
	XDONE : BOOL;
	XERROR : BOOL;
	EERRORID : L_IE1P_Error;
END_VAR
VAR
	XEXECUTEOLD : BOOL := FALSE;
END_VAR
END_FUNCTION_BLOCK

(* ---- L_MC1P_RESETHOMEPOSITION.pou ---- *)
FUNCTION_BLOCK L_MC1P_RESETHOMEPOSITION EXTENDS L_MC1P_Template
VAR_INPUT
	XEXECUTE : BOOL;
	XRESETPOSITIONOFFSET : BOOL;
END_VAR
VAR_OUTPUT
	XDONE : BOOL;
	XBUSY : BOOL;
	XERROR : BOOL;
	EERRORID : L_IE1P_Error;
END_VAR
VAR
	PAXIS : POINTER TO _AXIS_REF_REAL;
	XEXECUTEOLD : BOOL := FALSE;
	XBUSYOLD : BOOL := FALSE;
	XRESETOUTPUT : BOOL := FALSE;
END_VAR
END_FUNCTION_BLOCK
